// Mitsubishi GX Developer project: パレット移載装置   PLC: Q02

PROGRAM MAIN
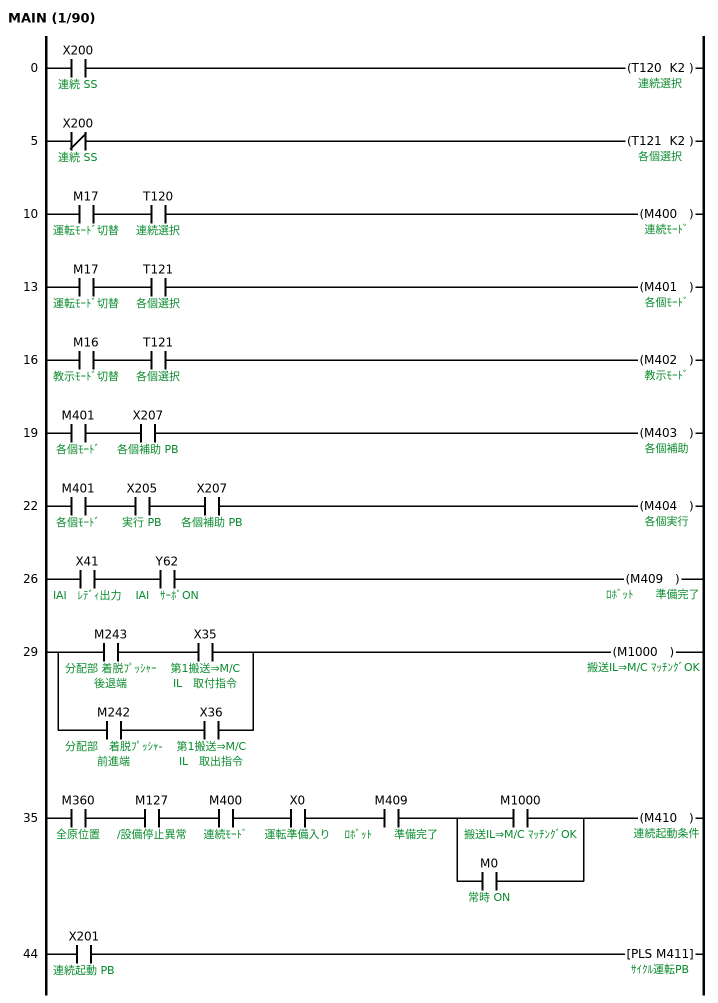
0     LD      X200  ; 連続 SS
      OUT     T120 K2  ; 連続選択
5     LDI     X200  ; 連続 SS
      OUT     T121 K2  ; 各個選択
10    LD      M17  ; 運転ﾓｰﾄﾞ切替
      AND     T120  ; 連続選択
      OUT     M400  ; 連続ﾓｰﾄﾞ
13    LD      M17  ; 運転ﾓｰﾄﾞ切替
      AND     T121  ; 各個選択
      OUT     M401  ; 各個ﾓｰﾄﾞ
16    LD      M16  ; 教示ﾓｰﾄﾞ切替
      AND     T121  ; 各個選択
      OUT     M402  ; 教示ﾓｰﾄﾞ
19    LD      M401  ; 各個ﾓｰﾄﾞ
      AND     X207  ; 各個補助 PB
      OUT     M403  ; 各個補助
22    LD      M401  ; 各個ﾓｰﾄﾞ
      AND     X205  ; 実行 PB
      AND     X207  ; 各個補助 PB
      OUT     M404  ; 各個実行
26    LD      X41  ; IAI　ﾚﾃﾞｨ出力
      AND     Y62  ; IAI　ｻｰﾎﾞON
      OUT     M409  ; ﾛﾎﾞｯﾄ　　準備完了
29    LD      M243  ; 分配部 着脱ﾌﾟｯｼｬｰ 後退端
      AND     X35  ; 第1搬送⇒M/C IL　取付指令
      LD      M242  ; 分配部　着脱ﾌﾟｯｼｬ- 前進端
      AND     X36  ; 第1搬送⇒M/C IL　取出指令
      ORB
      OUT     M1000  ; 搬送IL⇒M/C ﾏｯﾁﾝｸﾞOK
35    LD      M360  ; 全原位置
      AND     M127  ; /設備停止異常
      AND     M400  ; 連続ﾓｰﾄﾞ
      AND     X0  ; 運転準備入り
      AND     M409  ; ﾛﾎﾞｯﾄ　　準備完了
      LD      M1000  ; 搬送IL⇒M/C ﾏｯﾁﾝｸﾞOK
      OR      M0  ; 常時 ON
      ANB
      OUT     M410  ; 連続起動条件
44    LD      X201  ; 連続起動 PB
      PLS     M411  ; ｻｲｸﾙ運転PB
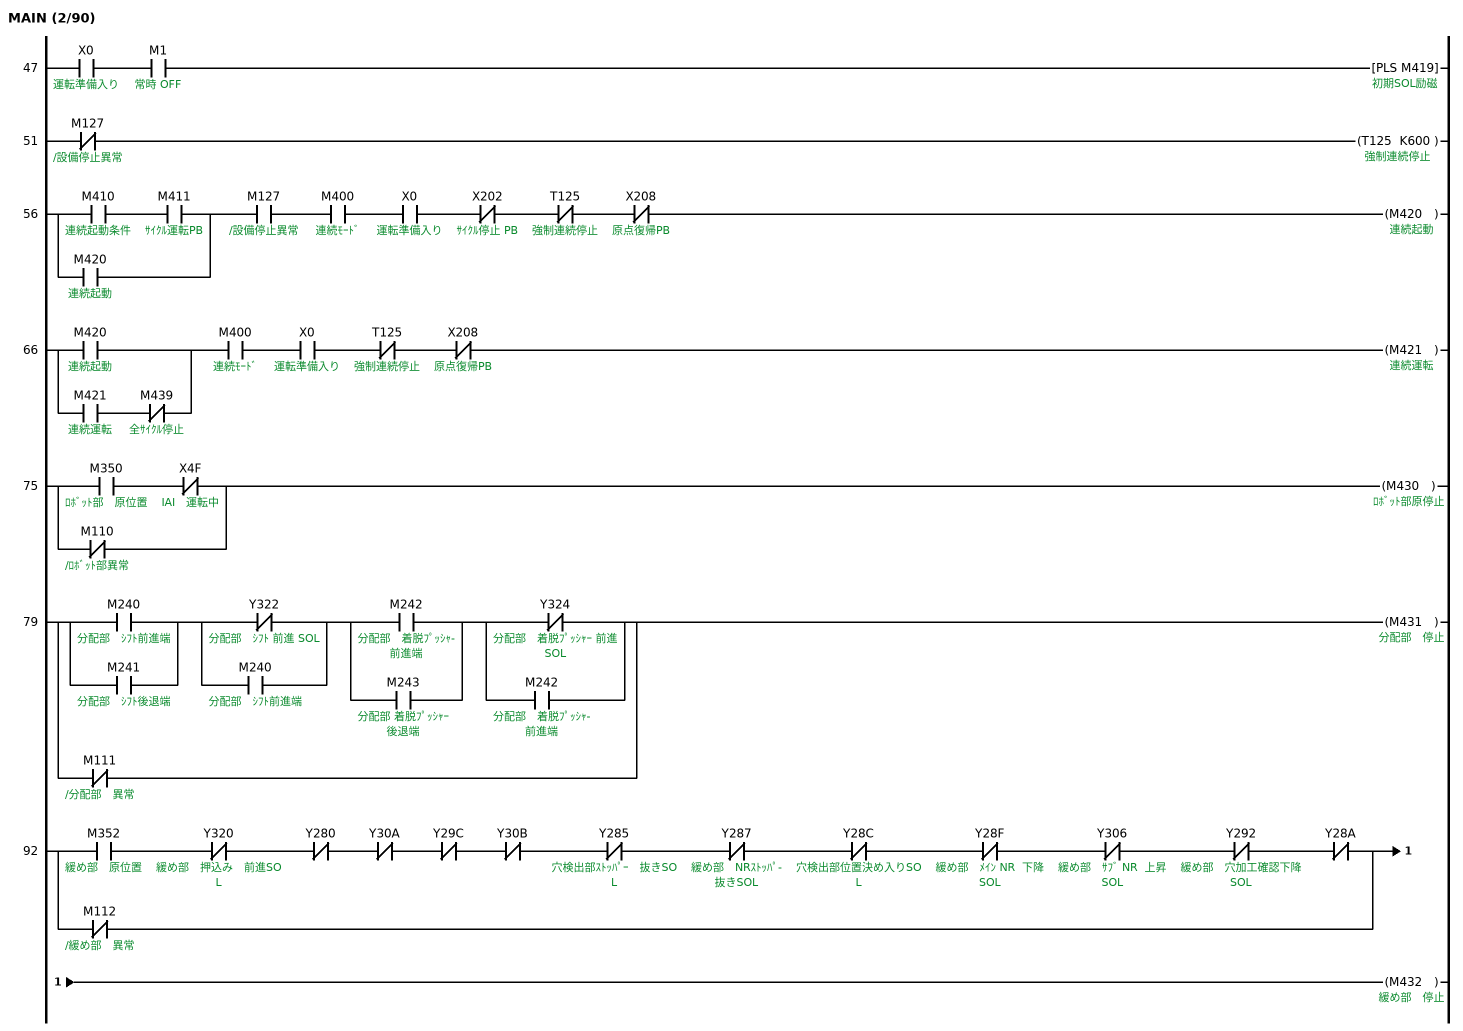
47    LD      X0  ; 運転準備入り
      AND     M1  ; 常時 OFF
      PLS     M419  ; 初期SOL励磁
51    LDI     M127  ; /設備停止異常
      OUT     T125 K600  ; 強制連続停止
56    LD      M410  ; 連続起動条件
      AND     M411  ; ｻｲｸﾙ運転PB
      OR      M420  ; 連続起動
      AND     M127  ; /設備停止異常
      AND     M400  ; 連続ﾓｰﾄﾞ
      AND     X0  ; 運転準備入り
      ANI     X202  ; ｻｲｸﾙ停止 PB
      ANI     T125  ; 強制連続停止
      ANI     X208  ; 原点復帰PB
      OUT     M420  ; 連続起動
66    LD      M420  ; 連続起動
      LD      M421  ; 連続運転
      ANI     M439  ; 全ｻｲｸﾙ停止
      ORB
      AND     M400  ; 連続ﾓｰﾄﾞ
      AND     X0  ; 運転準備入り
      ANI     T125  ; 強制連続停止
      ANI     X208  ; 原点復帰PB
      OUT     M421  ; 連続運転
75    LD      M350  ; ﾛﾎﾞｯﾄ部　原位置
      ANI     X4F  ; IAI　運転中
      ORI     M110  ; /ﾛﾎﾞｯﾄ部異常
      OUT     M430  ; ﾛﾎﾞｯﾄ部原停止
79    LD      M240  ; 分配部　ｼﾌﾄ前進端
      OR      M241  ; 分配部　ｼﾌﾄ後退端
      LDI     Y322  ; 分配部　ｼﾌﾄ 前進 SOL
      OR      M240  ; 分配部　ｼﾌﾄ前進端
      ANB
      LD      M242  ; 分配部　着脱ﾌﾟｯｼｬ- 前進端
      OR      M243  ; 分配部 着脱ﾌﾟｯｼｬｰ 後退端
      ANB
      LDI     Y324  ; 分配部　着脱ﾌﾟｯｼｬｰ 前進 SOL
      OR      M242  ; 分配部　着脱ﾌﾟｯｼｬ- 前進端
      ANB
      ORI     M111  ; /分配部　異常
      OUT     M431  ; 分配部　停止
92    LD      M352  ; 緩め部　原位置
      ANI     Y320  ; 緩め部　押込み　前進SOL
      ANI     Y280
      ANI     Y30A
      ANI     Y29C
      ANI     Y30B
      ANI     Y285  ; 穴検出部ｽﾄｯﾊﾟｰ　抜きSOL
      ANI     Y287  ; 緩め部　NRｽﾄｯﾊﾟ-抜きSOL
      ANI     Y28C  ; 穴検出部位置決め入りSOL
      ANI     Y28F  ; 緩め部　ﾒｲﾝ NR  下降 SOL
      ANI     Y306  ; 緩め部　ｻﾌﾞ NR  上昇 SOL
      ANI     Y292  ; 緩め部　穴加工確認下降 SOL
      ANI     Y28A
      ORI     M112  ; /緩め部　異常
      OUT     M432  ; 緩め部　停止
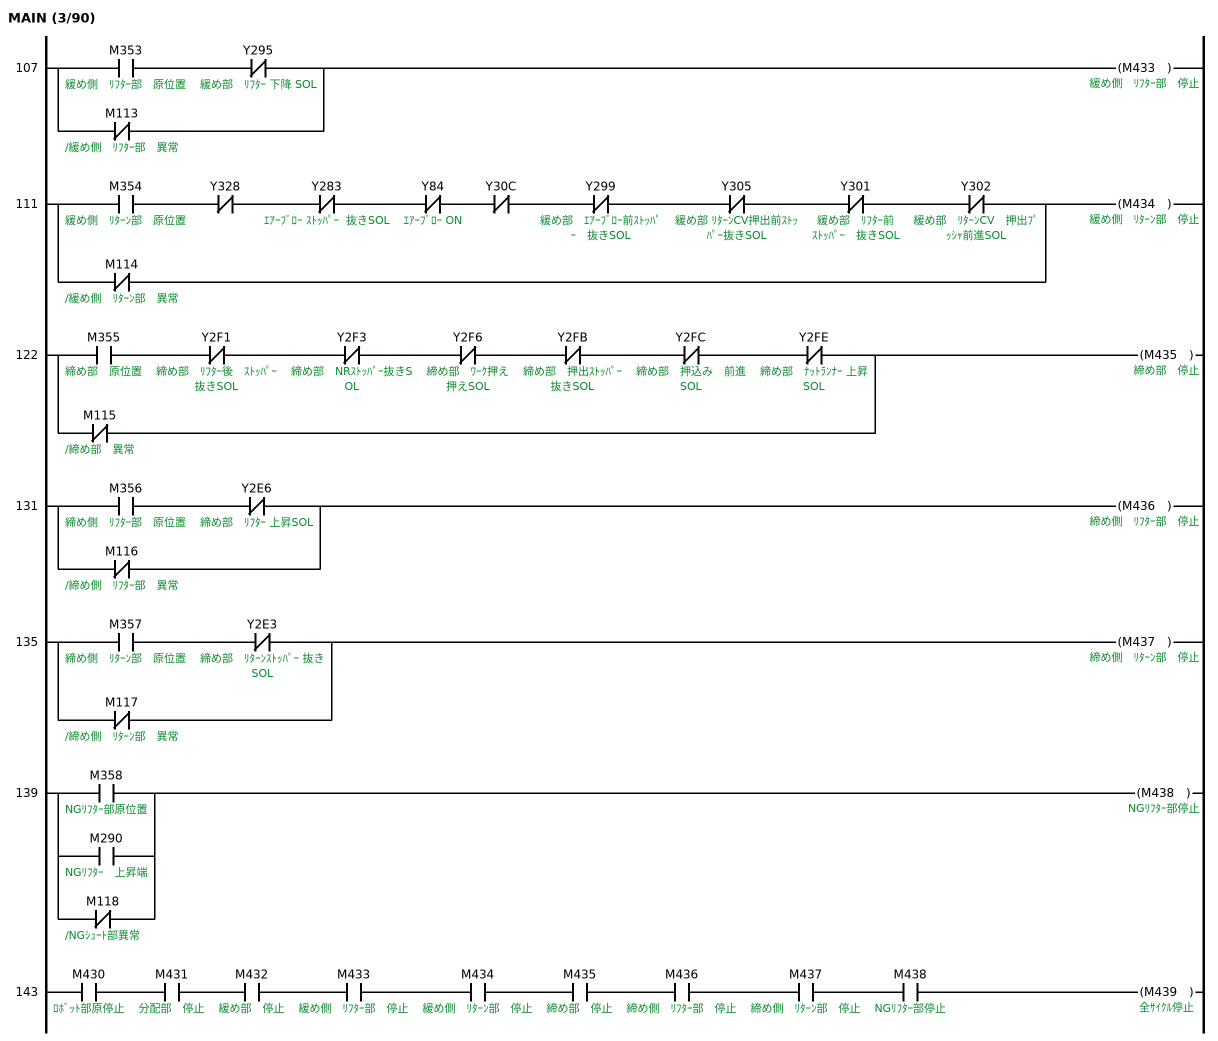
107   LD      M353  ; 緩め側　ﾘﾌﾀｰ部　原位置
      ANI     Y295  ; 緩め部　ﾘﾌﾀｰ 下降 SOL
      ORI     M113  ; /緩め側　ﾘﾌﾀｰ部　異常
      OUT     M433  ; 緩め側　ﾘﾌﾀｰ部　停止
111   LD      M354  ; 緩め側　ﾘﾀｰﾝ部　原位置
      ANI     Y328
      ANI     Y283  ; ｴｱｰﾌﾞﾛｰ ｽﾄｯﾊﾟｰ  抜きSOL
      ANI     Y84  ; ｴｱｰﾌﾞﾛｰ ON
      ANI     Y30C
      ANI     Y299  ; 緩め部　ｴｱｰﾌﾞﾛｰ前ｽﾄｯﾊﾟｰ　抜きSOL
      ANI     Y305  ; 緩め部 ﾘﾀｰﾝCV押出前ｽﾄｯﾊﾟｰ抜きSOL
      ANI     Y301  ; 緩め部　ﾘﾌﾀｰ前  ｽﾄｯﾊﾟｰ　抜きSOL
      ANI     Y302  ; 緩め部　ﾘﾀｰﾝCV　押出ﾌﾟｯｼｬ前進SOL
      ORI     M114  ; /緩め側　ﾘﾀｰﾝ部　異常
      OUT     M434  ; 緩め側　ﾘﾀｰﾝ部　停止
122   LD      M355  ; 締め部　原位置
      ANI     Y2F1  ; 締め部　ﾘﾌﾀｰ後　ｽﾄｯﾊﾟｰ　抜きSOL
      ANI     Y2F3  ; 締め部　NRｽﾄｯﾊﾟｰ抜きSOL
      ANI     Y2F6  ; 締め部　ﾜｰｸ押え 押えSOL
      ANI     Y2FB  ; 締め部　押出ｽﾄｯﾊﾟｰ 抜きSOL
      ANI     Y2FC  ; 締め部　押込み　前進 SOL
      ANI     Y2FE  ; 締め部　ﾅｯﾄﾗﾝﾅｰ 上昇 SOL
      ORI     M115  ; /締め部　異常
      OUT     M435  ; 締め部　停止
131   LD      M356  ; 締め側　ﾘﾌﾀｰ部　原位置
      ANI     Y2E6  ; 締め部　ﾘﾌﾀｰ 上昇SOL
      ORI     M116  ; /締め側　ﾘﾌﾀｰ部　異常
      OUT     M436  ; 締め側　ﾘﾌﾀｰ部　停止
135   LD      M357  ; 締め側　ﾘﾀｰﾝ部　原位置
      ANI     Y2E3  ; 締め部　ﾘﾀｰﾝｽﾄｯﾊﾟｰ 抜き SOL
      ORI     M117  ; /締め側　ﾘﾀｰﾝ部　異常
      OUT     M437  ; 締め側　ﾘﾀｰﾝ部　停止
139   LD      M358  ; NGﾘﾌﾀｰ部原位置
      OR      M290  ; NGﾘﾌﾀｰ　上昇端
      ORI     M118  ; /NGｼｭｰﾄ部異常
      OUT     M438  ; NGﾘﾌﾀｰ部停止
143   LD      M430  ; ﾛﾎﾞｯﾄ部原停止
      AND     M431  ; 分配部　停止
      AND     M432  ; 緩め部　停止
      AND     M433  ; 緩め側　ﾘﾌﾀｰ部　停止
      AND     M434  ; 緩め側　ﾘﾀｰﾝ部　停止
      AND     M435  ; 締め部　停止
      AND     M436  ; 締め側　ﾘﾌﾀｰ部　停止
      AND     M437  ; 締め側　ﾘﾀｰﾝ部　停止
      AND     M438  ; NGﾘﾌﾀｰ部停止
      OUT     M439  ; 全ｻｲｸﾙ停止
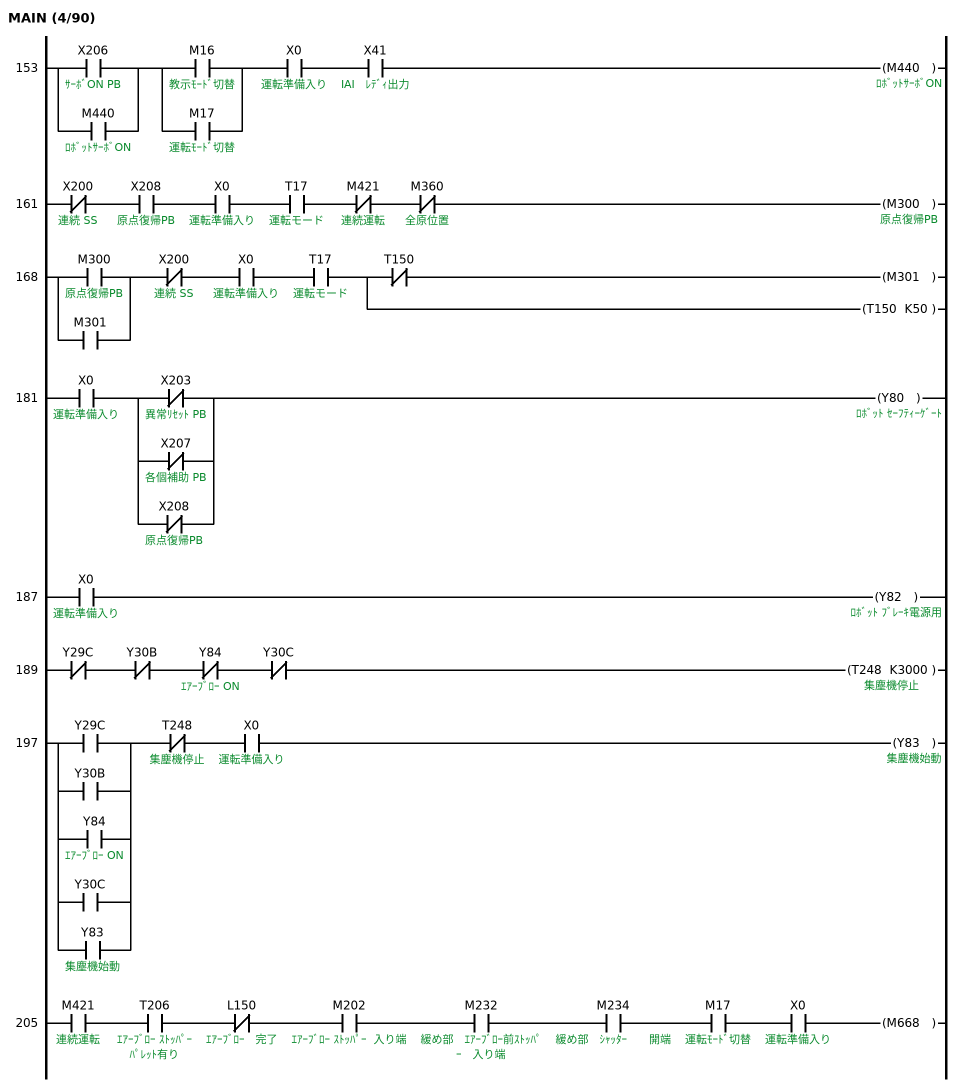
153   LD      X206  ; ｻｰﾎﾞON PB
      OR      M440  ; ﾛﾎﾞｯﾄｻｰﾎﾞON
      LD      M16  ; 教示ﾓｰﾄﾞ切替
      OR      M17  ; 運転ﾓｰﾄﾞ切替
      ANB
      AND     X0  ; 運転準備入り
      AND     X41  ; IAI　ﾚﾃﾞｨ出力
      OUT     M440  ; ﾛﾎﾞｯﾄｻｰﾎﾞON
161   LDI     X200  ; 連続 SS
      AND     X208  ; 原点復帰PB
      AND     X0  ; 運転準備入り
      AND     T17  ; 運転モード
      ANI     M421  ; 連続運転
      ANI     M360  ; 全原位置
      OUT     M300  ; 原点復帰PB
168   LD      M300  ; 原点復帰PB
      OR      M301
      ANI     X200  ; 連続 SS
      AND     X0  ; 運転準備入り
      AND     T17  ; 運転モード
      MPS
      ANI     T150
      OUT     M301
      MPP
      OUT     T150 K50
181   LD      X0  ; 運転準備入り
      LDI     X203  ; 異常ﾘｾｯﾄ PB
      ORI     X207  ; 各個補助 PB
      ORI     X208  ; 原点復帰PB
      ANB
      OUT     Y80  ; ﾛﾎﾞｯﾄ ｾｰﾌﾃｨｰｹﾞｰﾄ
187   LD      X0  ; 運転準備入り
      OUT     Y82  ; ﾛﾎﾞｯﾄ ﾌﾞﾚｰｷ電源用
189   LDI     Y29C
      ANI     Y30B
      ANI     Y84  ; ｴｱｰﾌﾞﾛｰ ON
      ANI     Y30C
      OUT     T248 K3000  ; 集塵機停止
197   LD      Y29C
      OR      Y30B
      OR      Y84  ; ｴｱｰﾌﾞﾛｰ ON
      OR      Y30C
      OR      Y83  ; 集塵機始動
      ANI     T248  ; 集塵機停止
      AND     X0  ; 運転準備入り
      OUT     Y83  ; 集塵機始動
205   LD      M421  ; 連続運転
      AND     T206  ; ｴｱｰﾌﾞﾛｰ ｽﾄｯﾊﾟｰ  ﾊﾟﾚｯﾄ有り
      ANI     L150  ; ｴｱｰﾌﾞﾛｰ　完了
      AND     M202  ; ｴｱｰﾌﾞﾛｰ ｽﾄｯﾊﾟｰ  入り端
      AND     M232  ; 緩め部　ｴｱｰﾌﾞﾛｰ前ｽﾄｯﾊﾟｰ　入り端
      AND     M234  ; 緩め部　ｼｬｯﾀｰ　　開端
      AND     M17  ; 運転ﾓｰﾄﾞ切替
      AND     X0  ; 運転準備入り
      OUT     M668
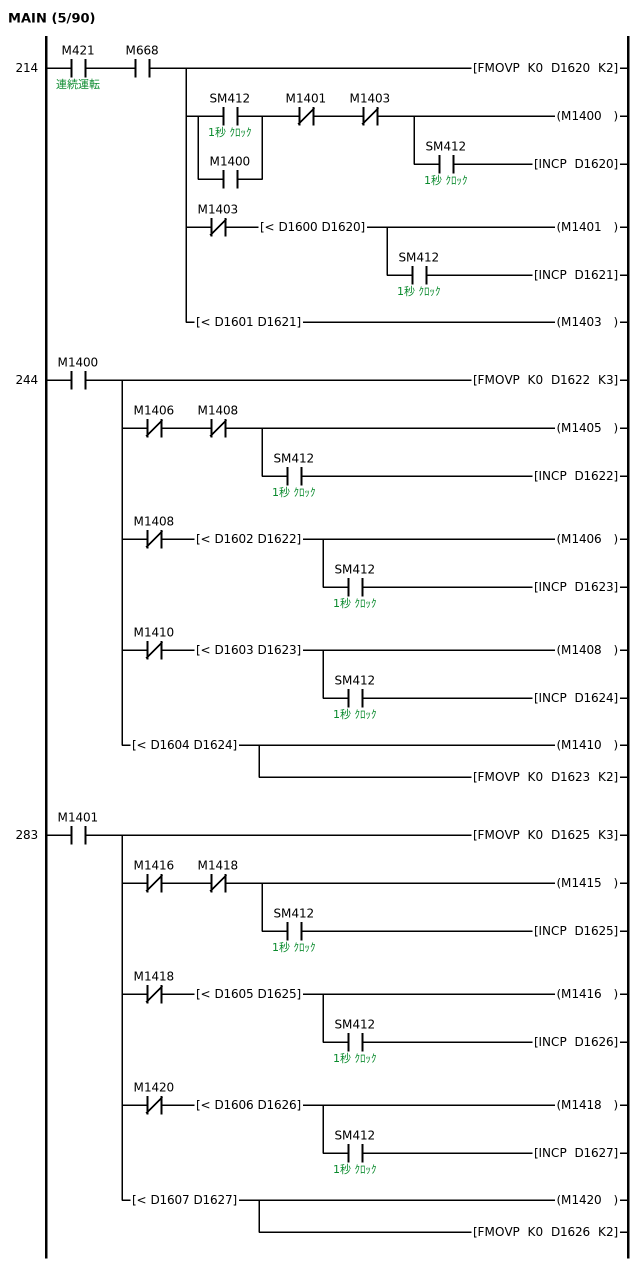
214   LD      M421  ; 連続運転
      AND     M668
      FMOVP   K0 D1620 K2
      MPS
      LD      SM412  ; 1秒 ｸﾛｯｸ
      OR      M1400
      ANB
      ANI     M1401
      ANI     M1403
      OUT     M1400
      AND     SM412  ; 1秒 ｸﾛｯｸ
      INCP    D1620
      MRD
      ANI     M1403
      AND<    D1600 D1620
      OUT     M1401
      AND     SM412  ; 1秒 ｸﾛｯｸ
      INCP    D1621
      MPP
      AND<    D1601 D1621
      OUT     M1403
244   LD      M1400
      FMOVP   K0 D1622 K3
      MPS
      ANI     M1406
      ANI     M1408
      OUT     M1405
      AND     SM412  ; 1秒 ｸﾛｯｸ
      INCP    D1622
      MRD
      ANI     M1408
      AND<    D1602 D1622
      OUT     M1406
      AND     SM412  ; 1秒 ｸﾛｯｸ
      INCP    D1623
      MRD
      ANI     M1410
      AND<    D1603 D1623
      OUT     M1408
      AND     SM412  ; 1秒 ｸﾛｯｸ
      INCP    D1624
      MPP
      AND<    D1604 D1624
      OUT     M1410
      FMOVP   K0 D1623 K2
283   LD      M1401
      FMOVP   K0 D1625 K3
      MPS
      ANI     M1416
      ANI     M1418
      OUT     M1415
      AND     SM412  ; 1秒 ｸﾛｯｸ
      INCP    D1625
      MRD
      ANI     M1418
      AND<    D1605 D1625
      OUT     M1416
      AND     SM412  ; 1秒 ｸﾛｯｸ
      INCP    D1626
      MRD
      ANI     M1420
      AND<    D1606 D1626
      OUT     M1418
      AND     SM412  ; 1秒 ｸﾛｯｸ
      INCP    D1627
      MPP
      AND<    D1607 D1627
      OUT     M1420
      FMOVP   K0 D1626 K2
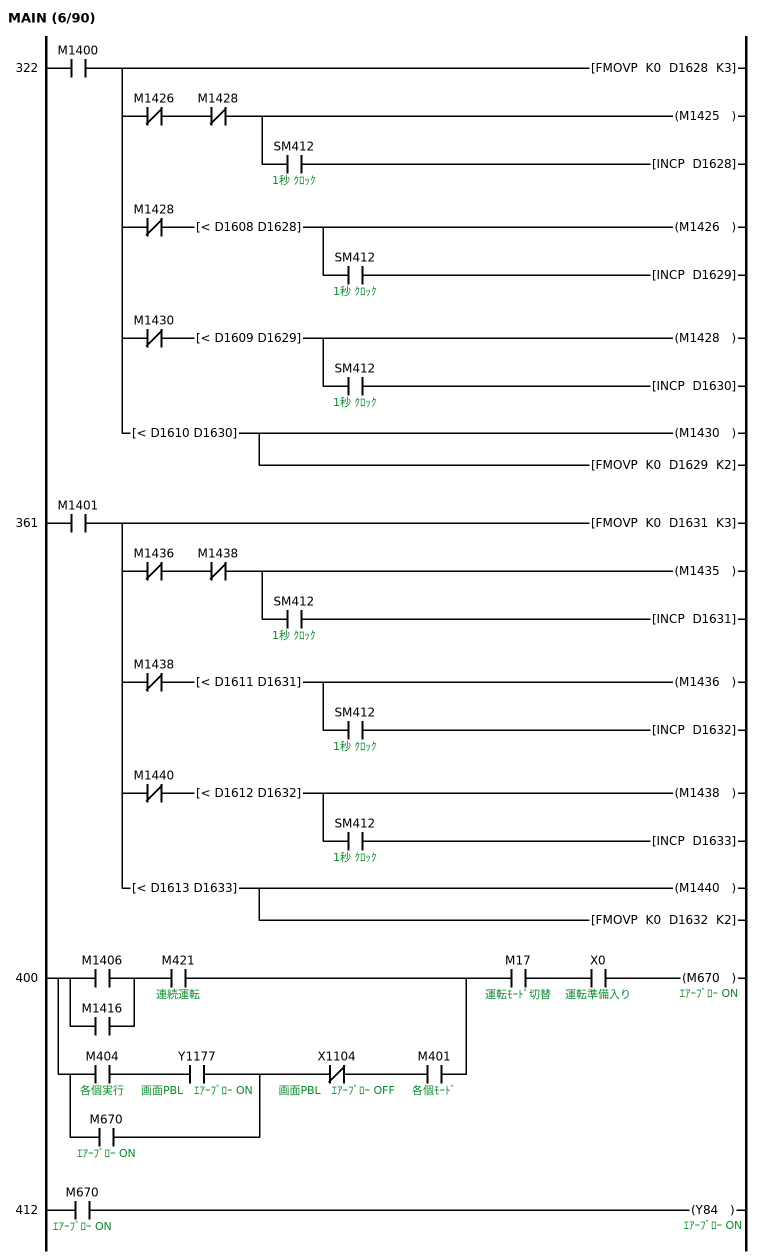
322   LD      M1400
      FMOVP   K0 D1628 K3
      MPS
      ANI     M1426
      ANI     M1428
      OUT     M1425
      AND     SM412  ; 1秒 ｸﾛｯｸ
      INCP    D1628
      MRD
      ANI     M1428
      AND<    D1608 D1628
      OUT     M1426
      AND     SM412  ; 1秒 ｸﾛｯｸ
      INCP    D1629
      MRD
      ANI     M1430
      AND<    D1609 D1629
      OUT     M1428
      AND     SM412  ; 1秒 ｸﾛｯｸ
      INCP    D1630
      MPP
      AND<    D1610 D1630
      OUT     M1430
      FMOVP   K0 D1629 K2
361   LD      M1401
      FMOVP   K0 D1631 K3
      MPS
      ANI     M1436
      ANI     M1438
      OUT     M1435
      AND     SM412  ; 1秒 ｸﾛｯｸ
      INCP    D1631
      MRD
      ANI     M1438
      AND<    D1611 D1631
      OUT     M1436
      AND     SM412  ; 1秒 ｸﾛｯｸ
      INCP    D1632
      MRD
      ANI     M1440
      AND<    D1612 D1632
      OUT     M1438
      AND     SM412  ; 1秒 ｸﾛｯｸ
      INCP    D1633
      MPP
      AND<    D1613 D1633
      OUT     M1440
      FMOVP   K0 D1632 K2
400   LD      M1406
      OR      M1416
      AND     M421  ; 連続運転
      LD      M404  ; 各個実行
      AND     Y1177  ; 画面PBL　ｴｱｰﾌﾞﾛｰ ON
      OR      M670  ; ｴｱｰﾌﾞﾛｰ ON
      ANI     X1104  ; 画面PBL　ｴｱｰﾌﾞﾛｰ OFF
      AND     M401  ; 各個ﾓｰﾄﾞ
      ORB
      AND     M17  ; 運転ﾓｰﾄﾞ切替
      AND     X0  ; 運転準備入り
      OUT     M670  ; ｴｱｰﾌﾞﾛｰ ON
412   LD      M670  ; ｴｱｰﾌﾞﾛｰ ON
      OUT     Y84  ; ｴｱｰﾌﾞﾛｰ ON
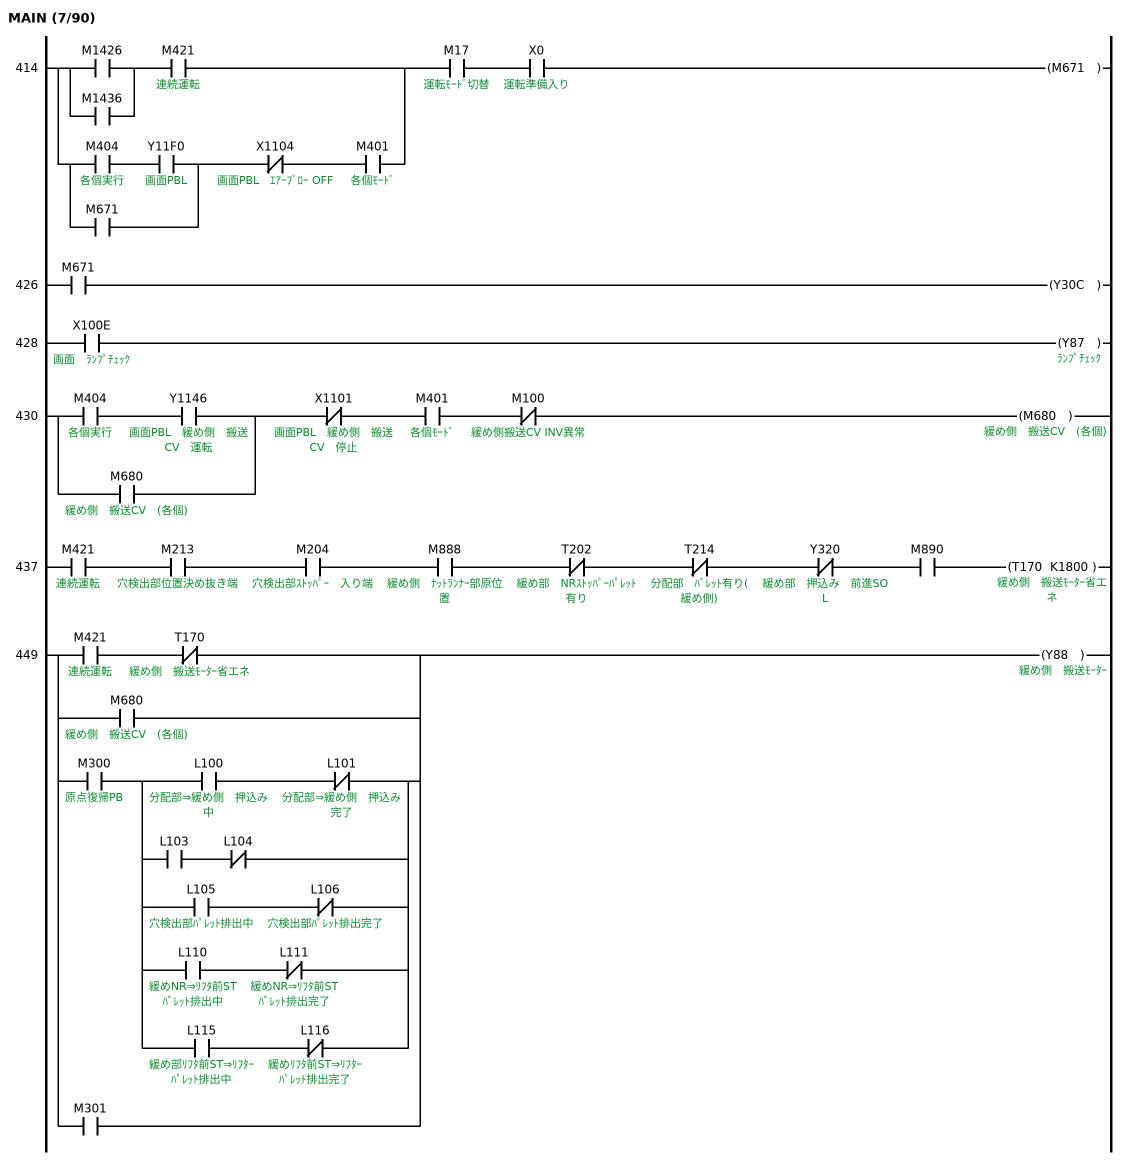
414   LD      M1426
      OR      M1436
      AND     M421  ; 連続運転
      LD      M404  ; 各個実行
      AND     Y11F0  ; 画面PBL
      OR      M671
      ANI     X1104  ; 画面PBL　ｴｱｰﾌﾞﾛｰ OFF
      AND     M401  ; 各個ﾓｰﾄﾞ
      ORB
      AND     M17  ; 運転ﾓｰﾄﾞ切替
      AND     X0  ; 運転準備入り
      OUT     M671
426   LD      M671
      OUT     Y30C
428   LD      X100E  ; 画面　ﾗﾝﾌﾟﾁｪｯｸ
      OUT     Y87  ; ﾗﾝﾌﾟﾁｪｯｸ
430   LD      M404  ; 各個実行
      AND     Y1146  ; 画面PBL　緩め側　搬送CV　運転
      OR      M680  ; 緩め側　搬送CV　(各個)
      ANI     X1101  ; 画面PBL　緩め側　搬送CV　停止
      AND     M401  ; 各個ﾓｰﾄﾞ
      ANI     M100  ; 緩め側搬送CV INV異常
      OUT     M680  ; 緩め側　搬送CV　(各個)
437   LD      M421  ; 連続運転
      AND     M213  ; 穴検出部位置決め抜き端
      AND     M204  ; 穴検出部ｽﾄｯﾊﾟｰ　入り端
      AND     M888  ; 緩め側　ﾅｯﾄﾗﾝﾅｰ部原位置
      ANI     T202  ; 緩め部　NRｽﾄｯﾊﾟｰﾊﾟﾚｯﾄ有り
      ANI     T214  ; 分配部　ﾊﾟﾚｯﾄ有り(緩め側)
      ANI     Y320  ; 緩め部　押込み　前進SOL
      AND     M890
      OUT     T170 K1800  ; 緩め側　搬送ﾓｰﾀｰ省エネ
449   LD      M421  ; 連続運転
      ANI     T170  ; 緩め側　搬送ﾓｰﾀｰ省エネ
      OR      M680  ; 緩め側　搬送CV　(各個)
      LD      M300  ; 原点復帰PB
      LD      L100  ; 分配部⇒緩め側　押込み中
      ANI     L101  ; 分配部⇒緩め側　押込み完了
      LD      L103
      ANI     L104
      ORB
      LD      L105  ; 穴検出部ﾊﾟﾚｯﾄ排出中
      ANI     L106  ; 穴検出部ﾊﾟﾚｯﾄ排出完了
      ORB
      LD      L110  ; 緩めNR⇒ﾘﾌﾀ前ST ﾊﾟﾚｯﾄ排出中
      ANI     L111  ; 緩めNR⇒ﾘﾌﾀ前ST ﾊﾟﾚｯﾄ排出完了
      ORB
      LD      L115  ; 緩め部ﾘﾌﾀ前ST⇒ﾘﾌﾀｰ ﾊﾟﾚｯﾄ排出中
      ANI     L116  ; 緩めﾘﾌﾀ前ST⇒ﾘﾌﾀｰ ﾊﾟﾚｯﾄ排出完了
      ORB
      ANB
      ORB
      OR      M301
      OUT     Y88  ; 緩め側　搬送ﾓｰﾀｰ
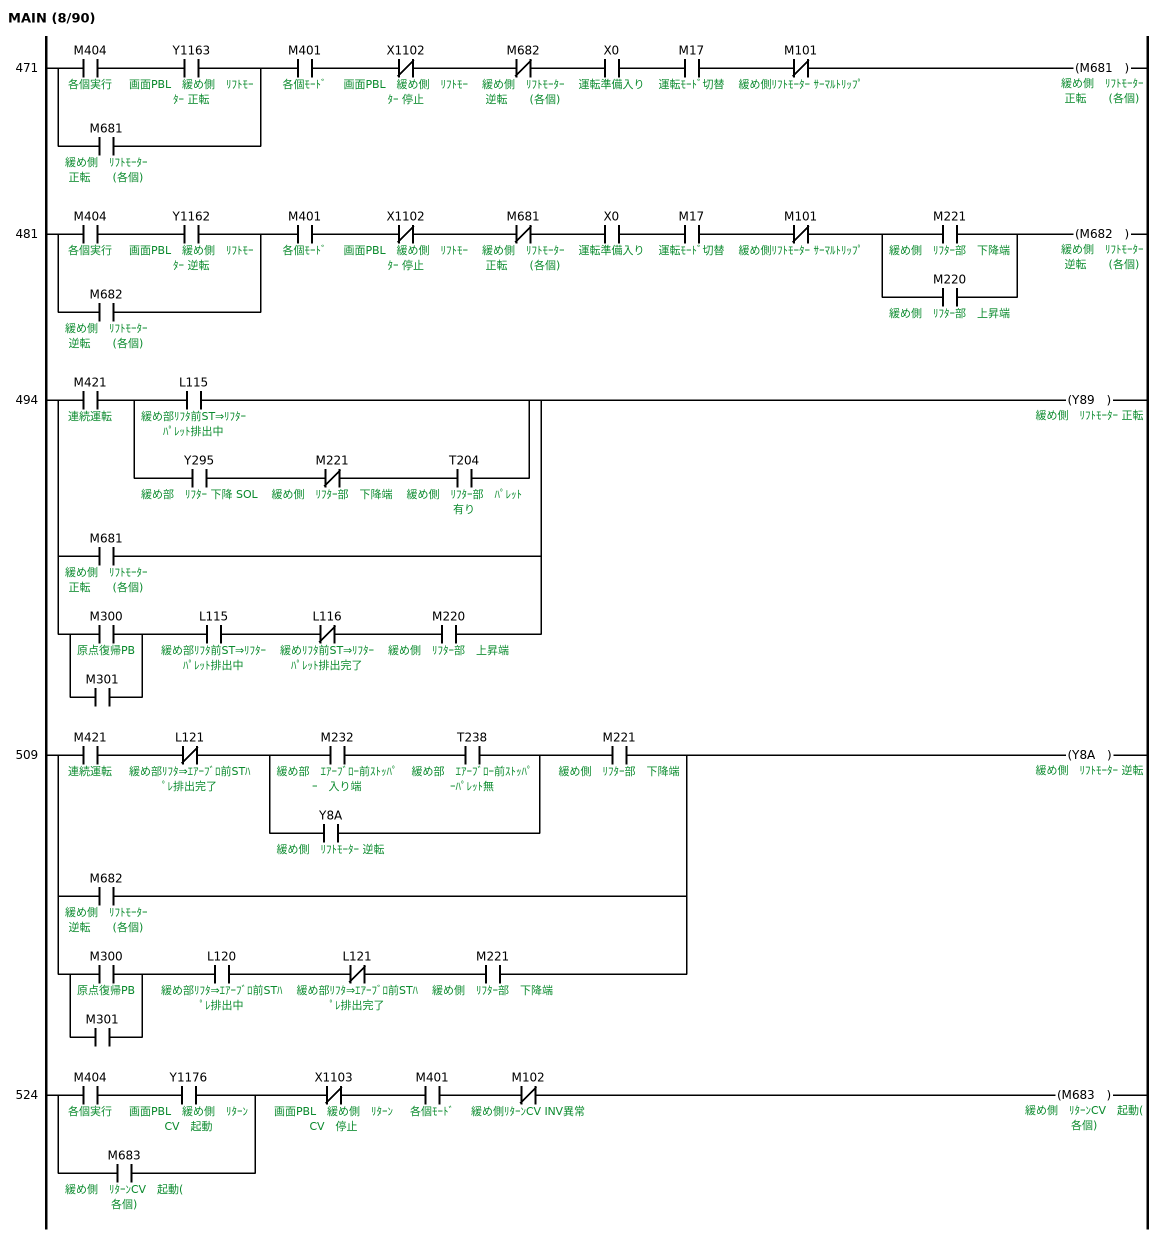
471   LD      M404  ; 各個実行
      AND     Y1163  ; 画面PBL　緩め側　ﾘﾌﾄﾓｰﾀｰ 正転
      OR      M681  ; 緩め側　ﾘﾌﾄﾓｰﾀｰ 正転　　(各個)
      AND     M401  ; 各個ﾓｰﾄﾞ
      ANI     X1102  ; 画面PBL　緩め側　ﾘﾌﾄﾓｰﾀｰ 停止
      ANI     M682  ; 緩め側　ﾘﾌﾄﾓｰﾀｰ 逆転　　(各個)
      AND     X0  ; 運転準備入り
      AND     M17  ; 運転ﾓｰﾄﾞ切替
      ANI     M101  ; 緩め側ﾘﾌﾄﾓｰﾀｰ ｻｰﾏﾙﾄﾘｯﾌﾟ
      OUT     M681  ; 緩め側　ﾘﾌﾄﾓｰﾀｰ 正転　　(各個)
481   LD      M404  ; 各個実行
      AND     Y1162  ; 画面PBL　緩め側　ﾘﾌﾄﾓｰﾀｰ 逆転
      OR      M682  ; 緩め側　ﾘﾌﾄﾓｰﾀｰ 逆転　　(各個)
      AND     M401  ; 各個ﾓｰﾄﾞ
      ANI     X1102  ; 画面PBL　緩め側　ﾘﾌﾄﾓｰﾀｰ 停止
      ANI     M681  ; 緩め側　ﾘﾌﾄﾓｰﾀｰ 正転　　(各個)
      AND     X0  ; 運転準備入り
      AND     M17  ; 運転ﾓｰﾄﾞ切替
      ANI     M101  ; 緩め側ﾘﾌﾄﾓｰﾀｰ ｻｰﾏﾙﾄﾘｯﾌﾟ
      LD      M221  ; 緩め側　ﾘﾌﾀｰ部　下降端
      OR      M220  ; 緩め側　ﾘﾌﾀｰ部　上昇端
      ANB
      OUT     M682  ; 緩め側　ﾘﾌﾄﾓｰﾀｰ 逆転　　(各個)
494   LD      M421  ; 連続運転
      LD      L115  ; 緩め部ﾘﾌﾀ前ST⇒ﾘﾌﾀｰ ﾊﾟﾚｯﾄ排出中
      LD      Y295  ; 緩め部　ﾘﾌﾀｰ 下降 SOL
      ANI     M221  ; 緩め側　ﾘﾌﾀｰ部　下降端
      AND     T204  ; 緩め側　ﾘﾌﾀｰ部　ﾊﾟﾚｯﾄ有り
      ORB
      ANB
      OR      M681  ; 緩め側　ﾘﾌﾄﾓｰﾀｰ 正転　　(各個)
      LD      M300  ; 原点復帰PB
      OR      M301
      AND     L115  ; 緩め部ﾘﾌﾀ前ST⇒ﾘﾌﾀｰ ﾊﾟﾚｯﾄ排出中
      ANI     L116  ; 緩めﾘﾌﾀ前ST⇒ﾘﾌﾀｰ ﾊﾟﾚｯﾄ排出完了
      AND     M220  ; 緩め側　ﾘﾌﾀｰ部　上昇端
      ORB
      OUT     Y89  ; 緩め側　ﾘﾌﾄﾓｰﾀｰ 正転
509   LD      M421  ; 連続運転
      ANI     L121  ; 緩め部ﾘﾌﾀ⇒ｴｱｰﾌﾞﾛ前STﾊﾟﾚ排出完了
      LD      M232  ; 緩め部　ｴｱｰﾌﾞﾛｰ前ｽﾄｯﾊﾟｰ　入り端
      AND     T238  ; 緩め部　ｴｱｰﾌﾞﾛｰ前ｽﾄｯﾊﾟｰﾊﾟﾚｯﾄ無
      OR      Y8A  ; 緩め側　ﾘﾌﾄﾓｰﾀｰ 逆転
      ANB
      AND     M221  ; 緩め側　ﾘﾌﾀｰ部　下降端
      OR      M682  ; 緩め側　ﾘﾌﾄﾓｰﾀｰ 逆転　　(各個)
      LD      M300  ; 原点復帰PB
      OR      M301
      AND     L120  ; 緩め部ﾘﾌﾀ⇒ｴｱｰﾌﾞﾛ前STﾊﾟﾚ排出中
      ANI     L121  ; 緩め部ﾘﾌﾀ⇒ｴｱｰﾌﾞﾛ前STﾊﾟﾚ排出完了
      AND     M221  ; 緩め側　ﾘﾌﾀｰ部　下降端
      ORB
      OUT     Y8A  ; 緩め側　ﾘﾌﾄﾓｰﾀｰ 逆転
524   LD      M404  ; 各個実行
      AND     Y1176  ; 画面PBL　緩め側　ﾘﾀｰﾝCV　起動
      OR      M683  ; 緩め側　ﾘﾀｰﾝCV　起動(各個)
      ANI     X1103  ; 画面PBL　緩め側　ﾘﾀｰﾝCV　停止
      AND     M401  ; 各個ﾓｰﾄﾞ
      ANI     M102  ; 緩め側ﾘﾀｰﾝCV INV異常
      OUT     M683  ; 緩め側　ﾘﾀｰﾝCV　起動(各個)
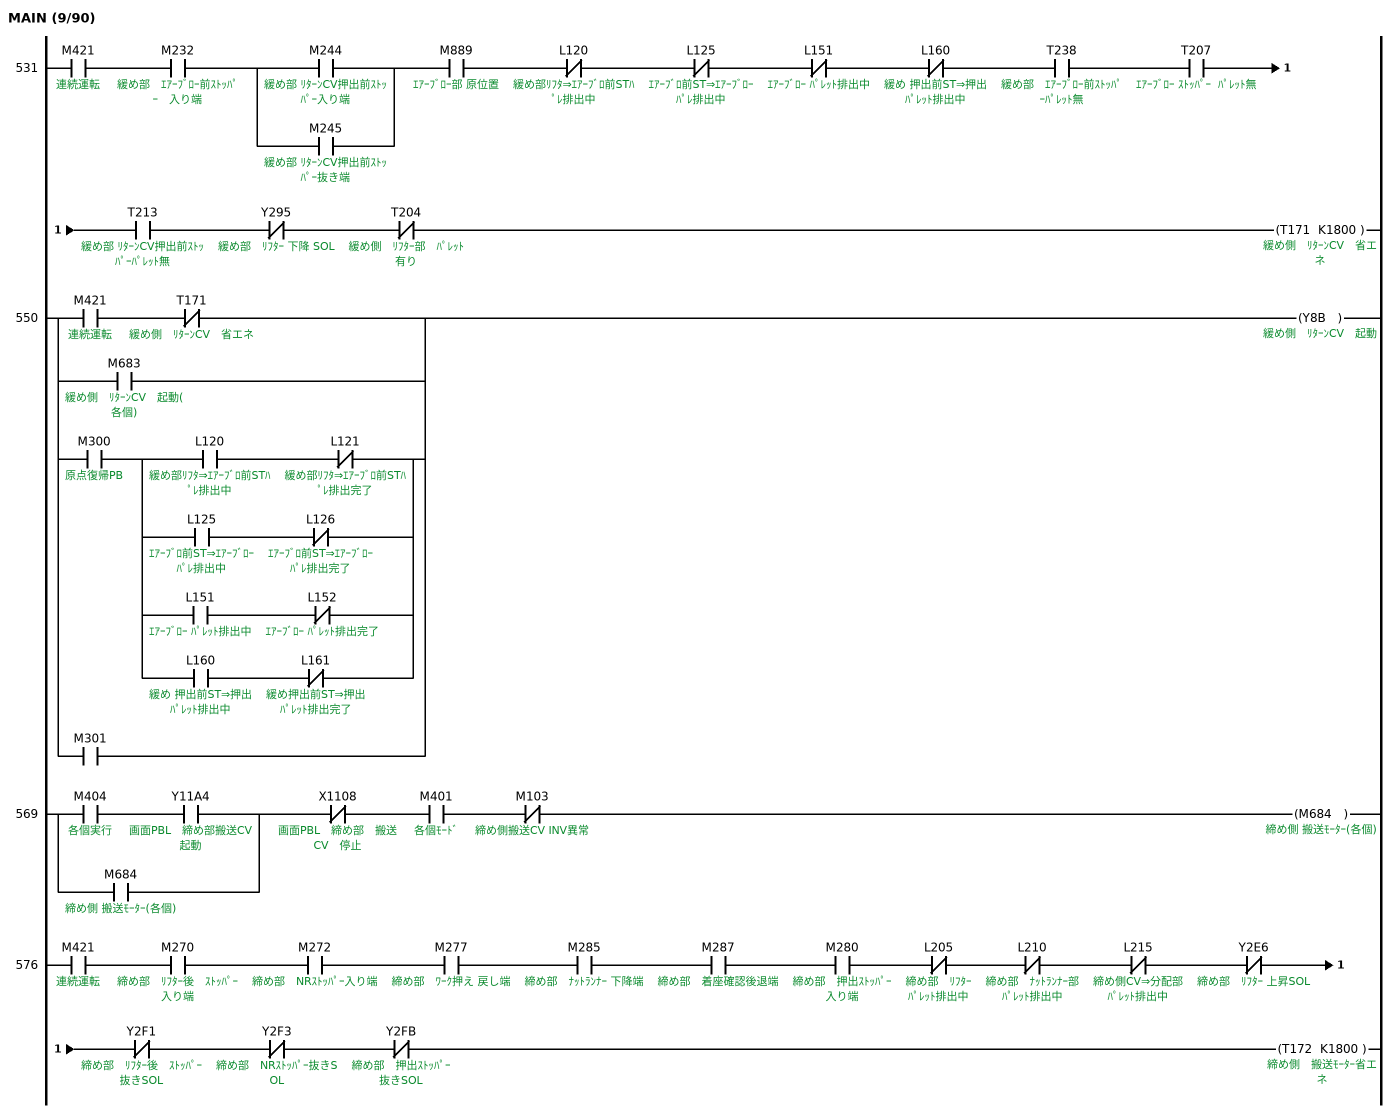
531   LD      M421  ; 連続運転
      AND     M232  ; 緩め部　ｴｱｰﾌﾞﾛｰ前ｽﾄｯﾊﾟｰ　入り端
      LD      M244  ; 緩め部 ﾘﾀｰﾝCV押出前ｽﾄｯﾊﾟｰ入り端
      OR      M245  ; 緩め部 ﾘﾀｰﾝCV押出前ｽﾄｯﾊﾟｰ抜き端
      ANB
      AND     M889  ; ｴｱｰﾌﾞﾛｰ部 原位置
      ANI     L120  ; 緩め部ﾘﾌﾀ⇒ｴｱｰﾌﾞﾛ前STﾊﾟﾚ排出中
      ANI     L125  ; ｴｱｰﾌﾞﾛ前ST⇒ｴｱｰﾌﾞﾛｰ ﾊﾟﾚ排出中
      ANI     L151  ; ｴｱｰﾌﾞﾛｰ ﾊﾟﾚｯﾄ排出中
      ANI     L160  ; 緩め 押出前ST⇒押出 ﾊﾟﾚｯﾄ排出中
      AND     T238  ; 緩め部　ｴｱｰﾌﾞﾛｰ前ｽﾄｯﾊﾟｰﾊﾟﾚｯﾄ無
      AND     T207  ; ｴｱｰﾌﾞﾛｰ ｽﾄｯﾊﾟｰ  ﾊﾟﾚｯﾄ無
      AND     T213  ; 緩め部 ﾘﾀｰﾝCV押出前ｽﾄｯﾊﾟｰﾊﾟﾚｯﾄ無
      ANI     Y295  ; 緩め部　ﾘﾌﾀｰ 下降 SOL
      ANI     T204  ; 緩め側　ﾘﾌﾀｰ部　ﾊﾟﾚｯﾄ有り
      OUT     T171 K1800  ; 緩め側　ﾘﾀｰﾝCV　省エネ
550   LD      M421  ; 連続運転
      ANI     T171  ; 緩め側　ﾘﾀｰﾝCV　省エネ
      OR      M683  ; 緩め側　ﾘﾀｰﾝCV　起動(各個)
      LD      M300  ; 原点復帰PB
      LD      L120  ; 緩め部ﾘﾌﾀ⇒ｴｱｰﾌﾞﾛ前STﾊﾟﾚ排出中
      ANI     L121  ; 緩め部ﾘﾌﾀ⇒ｴｱｰﾌﾞﾛ前STﾊﾟﾚ排出完了
      LD      L125  ; ｴｱｰﾌﾞﾛ前ST⇒ｴｱｰﾌﾞﾛｰ ﾊﾟﾚ排出中
      ANI     L126  ; ｴｱｰﾌﾞﾛ前ST⇒ｴｱｰﾌﾞﾛｰ ﾊﾟﾚ排出完了
      ORB
      LD      L151  ; ｴｱｰﾌﾞﾛｰ ﾊﾟﾚｯﾄ排出中
      ANI     L152  ; ｴｱｰﾌﾞﾛｰ ﾊﾟﾚｯﾄ排出完了
      ORB
      LD      L160  ; 緩め 押出前ST⇒押出 ﾊﾟﾚｯﾄ排出中
      ANI     L161  ; 緩め押出前ST⇒押出 ﾊﾟﾚｯﾄ排出完了
      ORB
      ANB
      ORB
      OR      M301
      OUT     Y8B  ; 緩め側　ﾘﾀｰﾝCV　起動
569   LD      M404  ; 各個実行
      AND     Y11A4  ; 画面PBL　締め部搬送CV起動
      OR      M684  ; 締め側 搬送ﾓｰﾀｰ(各個)
      ANI     X1108  ; 画面PBL　締め部　搬送CV　停止
      AND     M401  ; 各個ﾓｰﾄﾞ
      ANI     M103  ; 締め側搬送CV INV異常
      OUT     M684  ; 締め側 搬送ﾓｰﾀｰ(各個)
576   LD      M421  ; 連続運転
      AND     M270  ; 締め部　ﾘﾌﾀｰ後　ｽﾄｯﾊﾟｰ　入り端
      AND     M272  ; 締め部　NRｽﾄｯﾊﾟｰ入り端
      AND     M277  ; 締め部　ﾜｰｸ押え 戻し端
      AND     M285  ; 締め部　ﾅｯﾄﾗﾝﾅｰ 下降端
      AND     M287  ; 締め部　着座確認後退端
      AND     M280  ; 締め部　押出ｽﾄｯﾊﾟｰ 入り端
      ANI     L205  ; 締め部　ﾘﾌﾀｰ ﾊﾟﾚｯﾄ排出中
      ANI     L210  ; 締め部　ﾅｯﾄﾗﾝﾅｰ部 ﾊﾟﾚｯﾄ排出中
      ANI     L215  ; 締め側CV⇒分配部 ﾊﾟﾚｯﾄ排出中
      ANI     Y2E6  ; 締め部　ﾘﾌﾀｰ 上昇SOL
      ANI     Y2F1  ; 締め部　ﾘﾌﾀｰ後　ｽﾄｯﾊﾟｰ　抜きSOL
      ANI     Y2F3  ; 締め部　NRｽﾄｯﾊﾟｰ抜きSOL
      ANI     Y2FB  ; 締め部　押出ｽﾄｯﾊﾟｰ 抜きSOL
      OUT     T172 K1800  ; 締め側　搬送ﾓｰﾀｰ省エネ
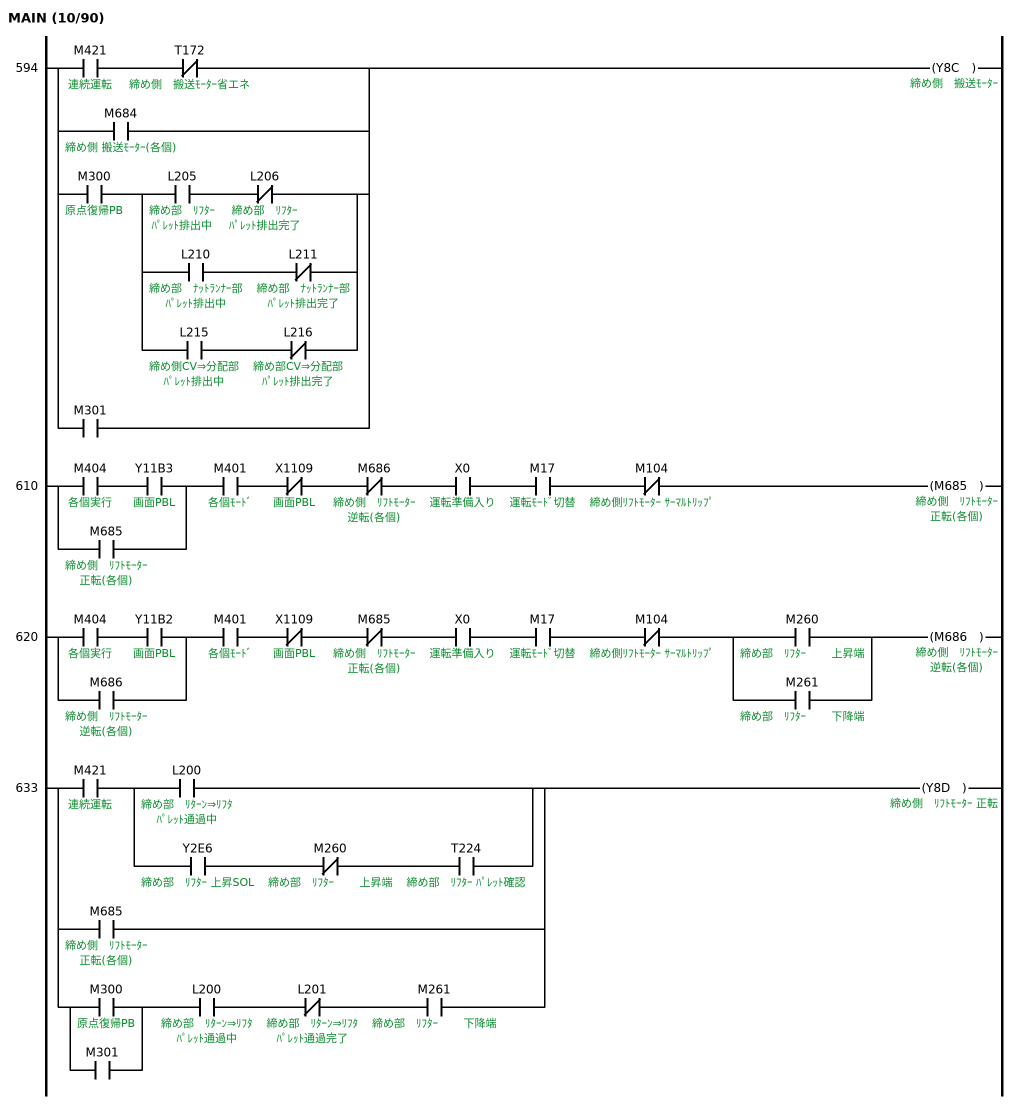
594   LD      M421  ; 連続運転
      ANI     T172  ; 締め側　搬送ﾓｰﾀｰ省エネ
      OR      M684  ; 締め側 搬送ﾓｰﾀｰ(各個)
      LD      M300  ; 原点復帰PB
      LD      L205  ; 締め部　ﾘﾌﾀｰ ﾊﾟﾚｯﾄ排出中
      ANI     L206  ; 締め部　ﾘﾌﾀｰ ﾊﾟﾚｯﾄ排出完了
      LD      L210  ; 締め部　ﾅｯﾄﾗﾝﾅｰ部 ﾊﾟﾚｯﾄ排出中
      ANI     L211  ; 締め部　ﾅｯﾄﾗﾝﾅｰ部 ﾊﾟﾚｯﾄ排出完了
      ORB
      LD      L215  ; 締め側CV⇒分配部 ﾊﾟﾚｯﾄ排出中
      ANI     L216  ; 締め部CV⇒分配部 ﾊﾟﾚｯﾄ排出完了
      ORB
      ANB
      ORB
      OR      M301
      OUT     Y8C  ; 締め側　搬送ﾓｰﾀｰ
610   LD      M404  ; 各個実行
      AND     Y11B3  ; 画面PBL
      OR      M685  ; 締め側　ﾘﾌﾄﾓｰﾀｰ 正転(各個)
      AND     M401  ; 各個ﾓｰﾄﾞ
      ANI     X1109  ; 画面PBL
      ANI     M686  ; 締め側　ﾘﾌﾄﾓｰﾀｰ 逆転(各個)
      AND     X0  ; 運転準備入り
      AND     M17  ; 運転ﾓｰﾄﾞ切替
      ANI     M104  ; 締め側ﾘﾌﾄﾓｰﾀｰ ｻｰﾏﾙﾄﾘｯﾌﾟ
      OUT     M685  ; 締め側　ﾘﾌﾄﾓｰﾀｰ 正転(各個)
620   LD      M404  ; 各個実行
      AND     Y11B2  ; 画面PBL
      OR      M686  ; 締め側　ﾘﾌﾄﾓｰﾀｰ 逆転(各個)
      AND     M401  ; 各個ﾓｰﾄﾞ
      ANI     X1109  ; 画面PBL
      ANI     M685  ; 締め側　ﾘﾌﾄﾓｰﾀｰ 正転(各個)
      AND     X0  ; 運転準備入り
      AND     M17  ; 運転ﾓｰﾄﾞ切替
      ANI     M104  ; 締め側ﾘﾌﾄﾓｰﾀｰ ｻｰﾏﾙﾄﾘｯﾌﾟ
      LD      M260  ; 締め部　ﾘﾌﾀｰ 　　上昇端
      OR      M261  ; 締め部　ﾘﾌﾀｰ 　　下降端
      ANB
      OUT     M686  ; 締め側　ﾘﾌﾄﾓｰﾀｰ 逆転(各個)
633   LD      M421  ; 連続運転
      LD      L200  ; 締め部　ﾘﾀｰﾝ⇒ﾘﾌﾀ ﾊﾟﾚｯﾄ通過中
      LD      Y2E6  ; 締め部　ﾘﾌﾀｰ 上昇SOL
      ANI     M260  ; 締め部　ﾘﾌﾀｰ 　　上昇端
      AND     T224  ; 締め部　ﾘﾌﾀｰ ﾊﾟﾚｯﾄ確認
      ORB
      ANB
      OR      M685  ; 締め側　ﾘﾌﾄﾓｰﾀｰ 正転(各個)
      LD      M300  ; 原点復帰PB
      OR      M301
      AND     L200  ; 締め部　ﾘﾀｰﾝ⇒ﾘﾌﾀ ﾊﾟﾚｯﾄ通過中
      ANI     L201  ; 締め部　ﾘﾀｰﾝ⇒ﾘﾌﾀ ﾊﾟﾚｯﾄ通過完了
      AND     M261  ; 締め部　ﾘﾌﾀｰ 　　下降端
      ORB
      OUT     Y8D  ; 締め側　ﾘﾌﾄﾓｰﾀｰ 正転
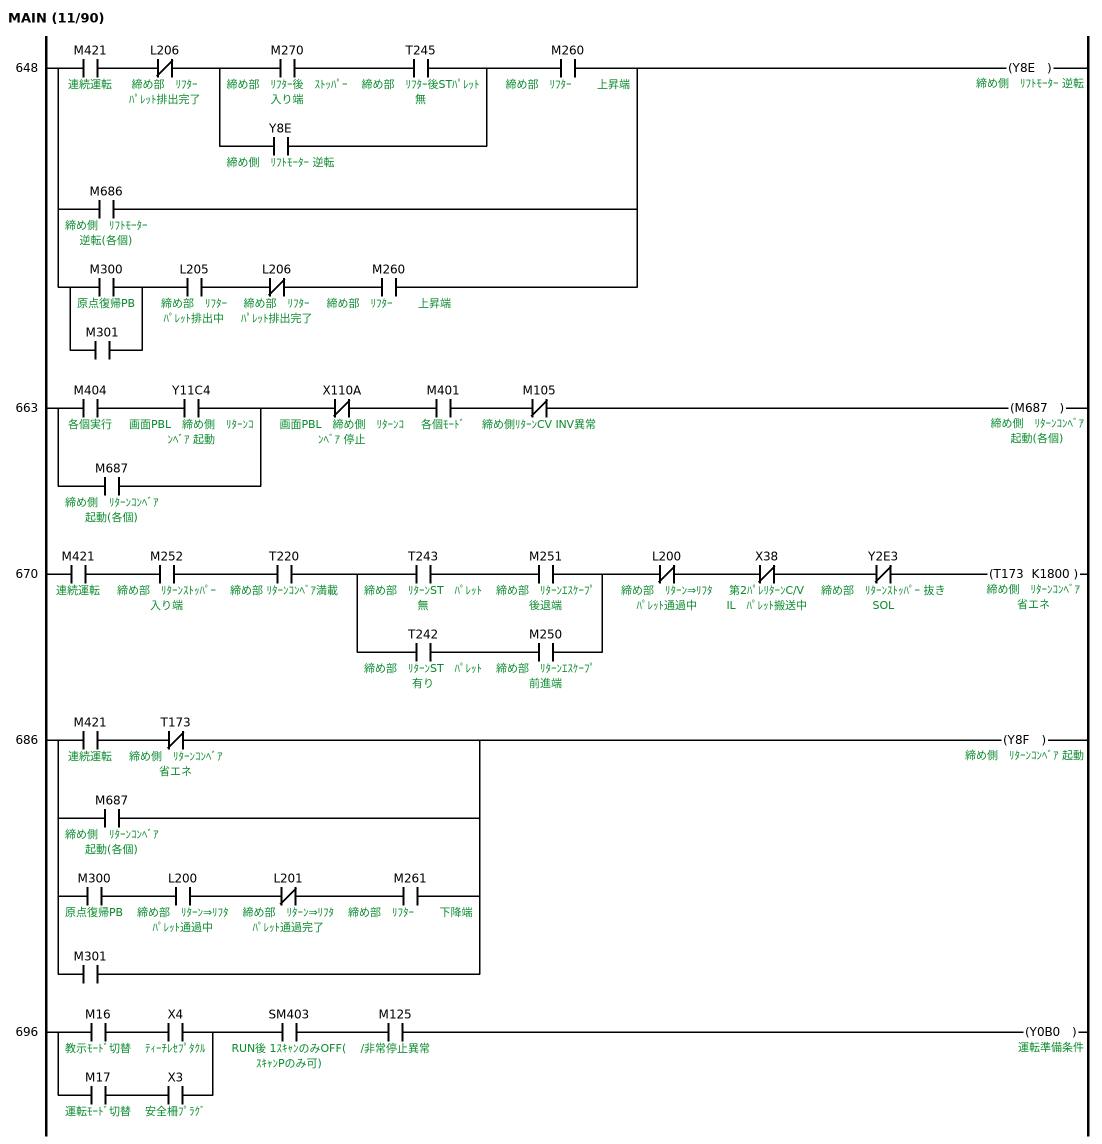
648   LD      M421  ; 連続運転
      ANI     L206  ; 締め部　ﾘﾌﾀｰ ﾊﾟﾚｯﾄ排出完了
      LD      M270  ; 締め部　ﾘﾌﾀｰ後　ｽﾄｯﾊﾟｰ　入り端
      AND     T245  ; 締め部　ﾘﾌﾀｰ後STﾊﾟﾚｯﾄ無
      OR      Y8E  ; 締め側　ﾘﾌﾄﾓｰﾀｰ 逆転
      ANB
      AND     M260  ; 締め部　ﾘﾌﾀｰ 　　上昇端
      OR      M686  ; 締め側　ﾘﾌﾄﾓｰﾀｰ 逆転(各個)
      LD      M300  ; 原点復帰PB
      OR      M301
      AND     L205  ; 締め部　ﾘﾌﾀｰ ﾊﾟﾚｯﾄ排出中
      ANI     L206  ; 締め部　ﾘﾌﾀｰ ﾊﾟﾚｯﾄ排出完了
      AND     M260  ; 締め部　ﾘﾌﾀｰ 　　上昇端
      ORB
      OUT     Y8E  ; 締め側　ﾘﾌﾄﾓｰﾀｰ 逆転
663   LD      M404  ; 各個実行
      AND     Y11C4  ; 画面PBL　締め側　ﾘﾀｰﾝｺﾝﾍﾞｱ 起動
      OR      M687  ; 締め側　ﾘﾀｰﾝｺﾝﾍﾞｱ 起動(各個)
      ANI     X110A  ; 画面PBL　締め側　ﾘﾀｰﾝｺﾝﾍﾞｱ 停止
      AND     M401  ; 各個ﾓｰﾄﾞ
      ANI     M105  ; 締め側ﾘﾀｰﾝCV INV異常
      OUT     M687  ; 締め側　ﾘﾀｰﾝｺﾝﾍﾞｱ 起動(各個)
670   LD      M421  ; 連続運転
      AND     M252  ; 締め部　ﾘﾀｰﾝｽﾄｯﾊﾟｰ 入り端
      AND     T220  ; 締め部 ﾘﾀｰﾝｺﾝﾍﾞｱ満載
      LD      T243  ; 締め部　ﾘﾀｰﾝST　ﾊﾟﾚｯﾄ無
      AND     M251  ; 締め部　ﾘﾀｰﾝｴｽｹｰﾌﾟ 後退端
      LD      T242  ; 締め部　ﾘﾀｰﾝST　ﾊﾟﾚｯﾄ有り
      AND     M250  ; 締め部　ﾘﾀｰﾝｴｽｹｰﾌﾟ 前進端
      ORB
      ANB
      ANI     L200  ; 締め部　ﾘﾀｰﾝ⇒ﾘﾌﾀ ﾊﾟﾚｯﾄ通過中
      ANI     X38  ; 第2ﾊﾟﾚﾘﾀｰﾝC/V IL　ﾊﾟﾚｯﾄ搬送中
      ANI     Y2E3  ; 締め部　ﾘﾀｰﾝｽﾄｯﾊﾟｰ 抜き SOL
      OUT     T173 K1800  ; 締め側　ﾘﾀｰﾝｺﾝﾍﾞｱ 省エネ
686   LD      M421  ; 連続運転
      ANI     T173  ; 締め側　ﾘﾀｰﾝｺﾝﾍﾞｱ 省エネ
      OR      M687  ; 締め側　ﾘﾀｰﾝｺﾝﾍﾞｱ 起動(各個)
      LD      M300  ; 原点復帰PB
      AND     L200  ; 締め部　ﾘﾀｰﾝ⇒ﾘﾌﾀ ﾊﾟﾚｯﾄ通過中
      ANI     L201  ; 締め部　ﾘﾀｰﾝ⇒ﾘﾌﾀ ﾊﾟﾚｯﾄ通過完了
      AND     M261  ; 締め部　ﾘﾌﾀｰ 　　下降端
      ORB
      OR      M301
      OUT     Y8F  ; 締め側　ﾘﾀｰﾝｺﾝﾍﾞｱ 起動
696   LD      M16  ; 教示ﾓｰﾄﾞ切替
      AND     X4  ; ﾃｨｰﾁﾚｾﾌﾟﾀｸﾙ
      LD      M17  ; 運転ﾓｰﾄﾞ切替
      AND     X3  ; 安全柵ﾌﾟﾗｸﾞ
      ORB
      AND     SM403  ; RUN後 1ｽｷｬﾝのみOFF(ｽｷｬﾝPのみ可)
      AND     M125  ; /非常停止異常
      OUT     Y0B0  ; 運転準備条件
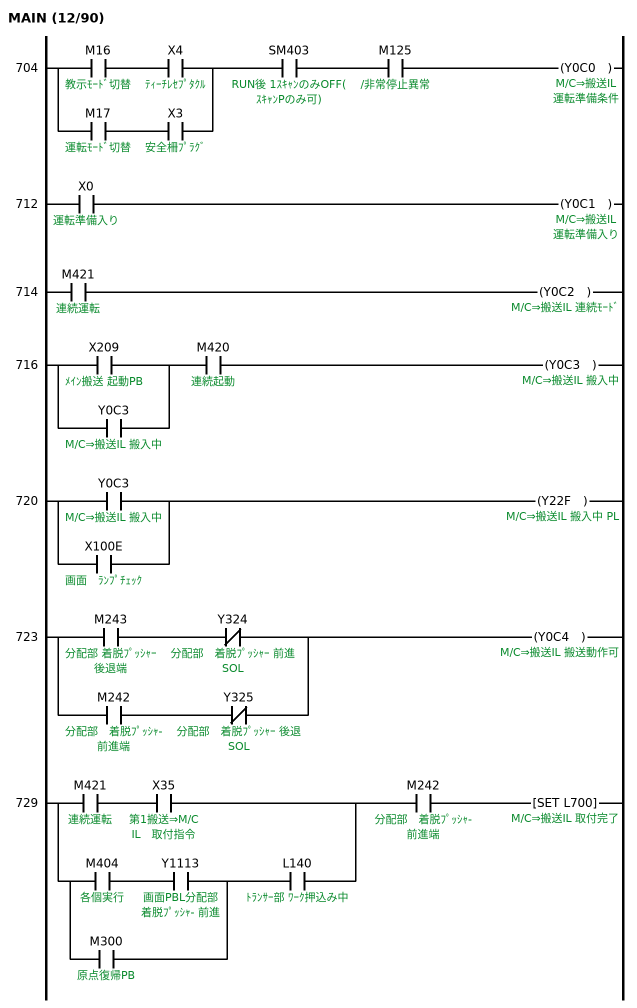
704   LD      M16  ; 教示ﾓｰﾄﾞ切替
      AND     X4  ; ﾃｨｰﾁﾚｾﾌﾟﾀｸﾙ
      LD      M17  ; 運転ﾓｰﾄﾞ切替
      AND     X3  ; 安全柵ﾌﾟﾗｸﾞ
      ORB
      AND     SM403  ; RUN後 1ｽｷｬﾝのみOFF(ｽｷｬﾝPのみ可)
      AND     M125  ; /非常停止異常
      OUT     Y0C0  ; M/C⇒搬送IL 運転準備条件
712   LD      X0  ; 運転準備入り
      OUT     Y0C1  ; M/C⇒搬送IL 運転準備入り
714   LD      M421  ; 連続運転
      OUT     Y0C2  ; M/C⇒搬送IL 連続ﾓｰﾄﾞ
716   LD      X209  ; ﾒｲﾝ搬送 起動PB
      OR      Y0C3  ; M/C⇒搬送IL 搬入中
      AND     M420  ; 連続起動
      OUT     Y0C3  ; M/C⇒搬送IL 搬入中
720   LD      Y0C3  ; M/C⇒搬送IL 搬入中
      OR      X100E  ; 画面　ﾗﾝﾌﾟﾁｪｯｸ
      OUT     Y22F  ; M/C⇒搬送IL 搬入中 PL
723   LD      M243  ; 分配部 着脱ﾌﾟｯｼｬｰ 後退端
      ANI     Y324  ; 分配部　着脱ﾌﾟｯｼｬｰ 前進 SOL
      LD      M242  ; 分配部　着脱ﾌﾟｯｼｬ- 前進端
      ANI     Y325  ; 分配部　着脱ﾌﾟｯｼｬｰ 後退 SOL
      ORB
      OUT     Y0C4  ; M/C⇒搬送IL 搬送動作可
729   LD      M421  ; 連続運転
      AND     X35  ; 第1搬送⇒M/C IL　取付指令
      LD      M404  ; 各個実行
      AND     Y1113  ; 画面PBL分配部 着脱ﾌﾟｯｼｬ- 前進
      OR      M300  ; 原点復帰PB
      AND     L140  ; ﾄﾗﾝｻｰ部 ﾜｰｸ押込み中
      ORB
      AND     M242  ; 分配部　着脱ﾌﾟｯｼｬ- 前進端
      SET     L700  ; M/C⇒搬送IL 取付完了
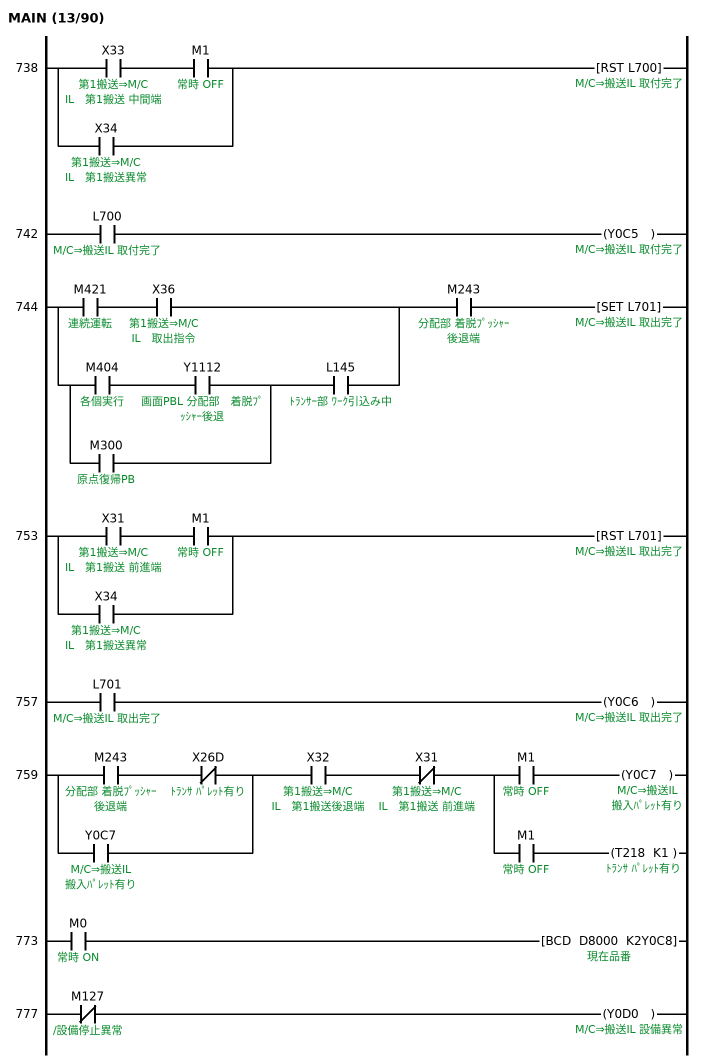
738   LD      X33  ; 第1搬送⇒M/C IL　第1搬送 中間端
      AND     M1  ; 常時 OFF
      OR      X34  ; 第1搬送⇒M/C IL　第1搬送異常
      RST     L700  ; M/C⇒搬送IL 取付完了
742   LD      L700  ; M/C⇒搬送IL 取付完了
      OUT     Y0C5  ; M/C⇒搬送IL 取付完了
744   LD      M421  ; 連続運転
      AND     X36  ; 第1搬送⇒M/C IL　取出指令
      LD      M404  ; 各個実行
      AND     Y1112  ; 画面PBL 分配部　着脱ﾌﾟｯｼｬｰ後退
      OR      M300  ; 原点復帰PB
      AND     L145  ; ﾄﾗﾝｻｰ部 ﾜｰｸ引込み中
      ORB
      AND     M243  ; 分配部 着脱ﾌﾟｯｼｬｰ 後退端
      SET     L701  ; M/C⇒搬送IL 取出完了
753   LD      X31  ; 第1搬送⇒M/C IL　第1搬送 前進端
      AND     M1  ; 常時 OFF
      OR      X34  ; 第1搬送⇒M/C IL　第1搬送異常
      RST     L701  ; M/C⇒搬送IL 取出完了
757   LD      L701  ; M/C⇒搬送IL 取出完了
      OUT     Y0C6  ; M/C⇒搬送IL 取出完了
759   LD      M243  ; 分配部 着脱ﾌﾟｯｼｬｰ 後退端
      ANI     X26D  ; ﾄﾗﾝｻ ﾊﾟﾚｯﾄ有り
      OR      Y0C7  ; M/C⇒搬送IL 搬入ﾊﾟﾚｯﾄ有り
      AND     X32  ; 第1搬送⇒M/C IL　第1搬送後退端
      ANI     X31  ; 第1搬送⇒M/C IL　第1搬送 前進端
      MPS
      AND     M1  ; 常時 OFF
      OUT     Y0C7  ; M/C⇒搬送IL 搬入ﾊﾟﾚｯﾄ有り
      MPP
      AND     M1  ; 常時 OFF
      OUT     T218 K1  ; ﾄﾗﾝｻ ﾊﾟﾚｯﾄ有り
773   LD      M0  ; 常時 ON
      BCD     D8000 K2Y0C8  ; 現在品番 / M/C⇒搬送IL ID情報 BCD01
777   LDI     M127  ; /設備停止異常
      OUT     Y0D0  ; M/C⇒搬送IL 設備異常
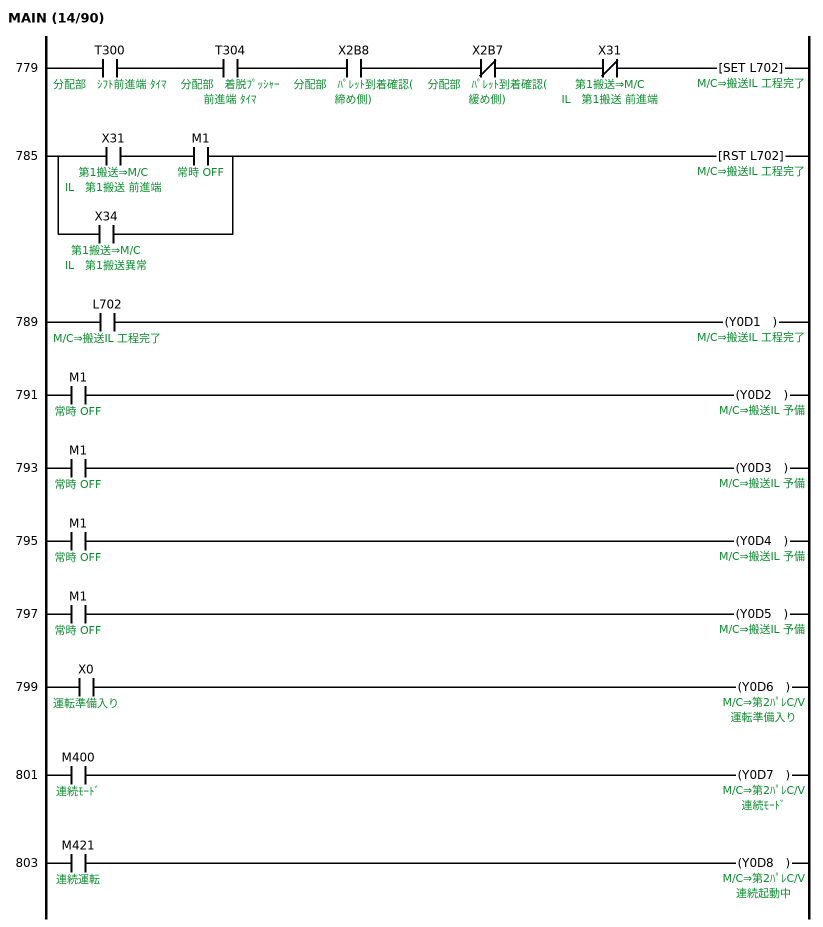
779   LD      T300  ; 分配部　ｼﾌﾄ前進端 ﾀｲﾏ
      AND     T304  ; 分配部　着脱ﾌﾟｯｼｬｰ 前進端 ﾀｲﾏ
      AND     X2B8  ; 分配部　ﾊﾟﾚｯﾄ到着確認(締め側)
      ANI     X2B7  ; 分配部　ﾊﾟﾚｯﾄ到着確認(緩め側)
      ANI     X31  ; 第1搬送⇒M/C IL　第1搬送 前進端
      SET     L702  ; M/C⇒搬送IL 工程完了
785   LD      X31  ; 第1搬送⇒M/C IL　第1搬送 前進端
      AND     M1  ; 常時 OFF
      OR      X34  ; 第1搬送⇒M/C IL　第1搬送異常
      RST     L702  ; M/C⇒搬送IL 工程完了
789   LD      L702  ; M/C⇒搬送IL 工程完了
      OUT     Y0D1  ; M/C⇒搬送IL 工程完了
791   LD      M1  ; 常時 OFF
      OUT     Y0D2  ; M/C⇒搬送IL 予備
793   LD      M1  ; 常時 OFF
      OUT     Y0D3  ; M/C⇒搬送IL 予備
795   LD      M1  ; 常時 OFF
      OUT     Y0D4  ; M/C⇒搬送IL 予備
797   LD      M1  ; 常時 OFF
      OUT     Y0D5  ; M/C⇒搬送IL 予備
799   LD      X0  ; 運転準備入り
      OUT     Y0D6  ; M/C⇒第2ﾊﾟﾚC/V 運転準備入り
801   LD      M400  ; 連続ﾓｰﾄﾞ
      OUT     Y0D7  ; M/C⇒第2ﾊﾟﾚC/V 連続ﾓｰﾄﾞ
803   LD      M421  ; 連続運転
      OUT     Y0D8  ; M/C⇒第2ﾊﾟﾚC/V 連続起動中
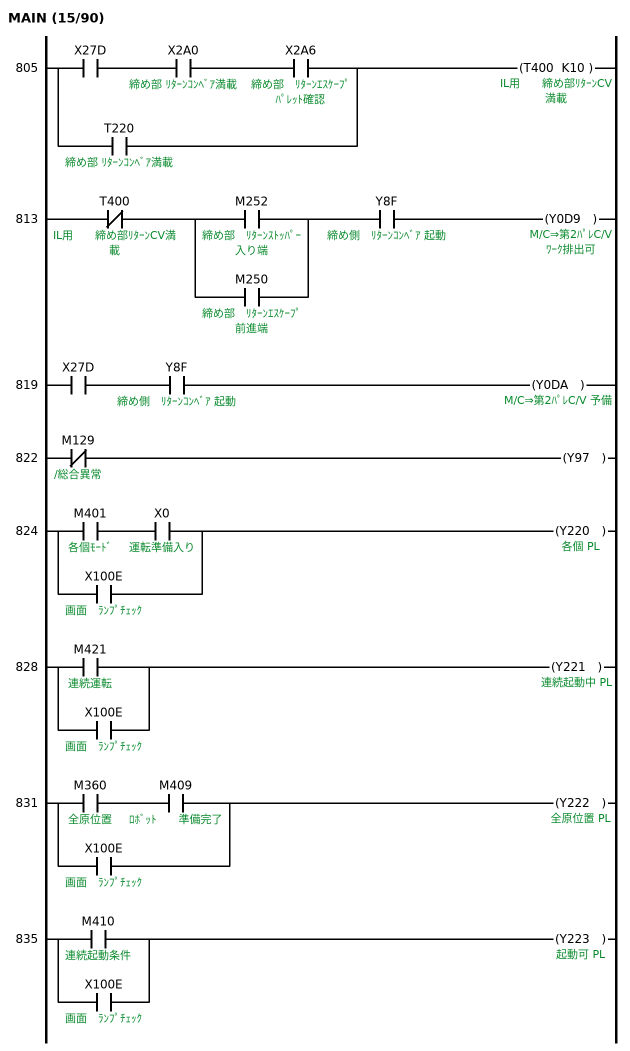
805   LD      X27D
      AND     X2A0  ; 締め部 ﾘﾀｰﾝｺﾝﾍﾞｱ満載
      AND     X2A6  ; 締め部　ﾘﾀｰﾝｴｽｹｰﾌﾟ ﾊﾟﾚｯﾄ確認
      OR      T220  ; 締め部 ﾘﾀｰﾝｺﾝﾍﾞｱ満載
      OUT     T400 K10  ; IL用　　締め部ﾘﾀｰﾝCV満載
813   LDI     T400  ; IL用　　締め部ﾘﾀｰﾝCV満載
      LD      M252  ; 締め部　ﾘﾀｰﾝｽﾄｯﾊﾟｰ 入り端
      OR      M250  ; 締め部　ﾘﾀｰﾝｴｽｹｰﾌﾟ 前進端
      ANB
      AND     Y8F  ; 締め側　ﾘﾀｰﾝｺﾝﾍﾞｱ 起動
      OUT     Y0D9  ; M/C⇒第2ﾊﾟﾚC/V ﾜｰｸ排出可
819   LD      X27D
      AND     Y8F  ; 締め側　ﾘﾀｰﾝｺﾝﾍﾞｱ 起動
      OUT     Y0DA  ; M/C⇒第2ﾊﾟﾚC/V 予備
822   LDI     M129  ; /総合異常
      OUT     Y97
824   LD      M401  ; 各個ﾓｰﾄﾞ
      AND     X0  ; 運転準備入り
      OR      X100E  ; 画面　ﾗﾝﾌﾟﾁｪｯｸ
      OUT     Y220  ; 各個 PL
828   LD      M421  ; 連続運転
      OR      X100E  ; 画面　ﾗﾝﾌﾟﾁｪｯｸ
      OUT     Y221  ; 連続起動中 PL
831   LD      M360  ; 全原位置
      AND     M409  ; ﾛﾎﾞｯﾄ　　準備完了
      OR      X100E  ; 画面　ﾗﾝﾌﾟﾁｪｯｸ
      OUT     Y222  ; 全原位置 PL
835   LD      M410  ; 連続起動条件
      OR      X100E  ; 画面　ﾗﾝﾌﾟﾁｪｯｸ
      OUT     Y223  ; 起動可 PL
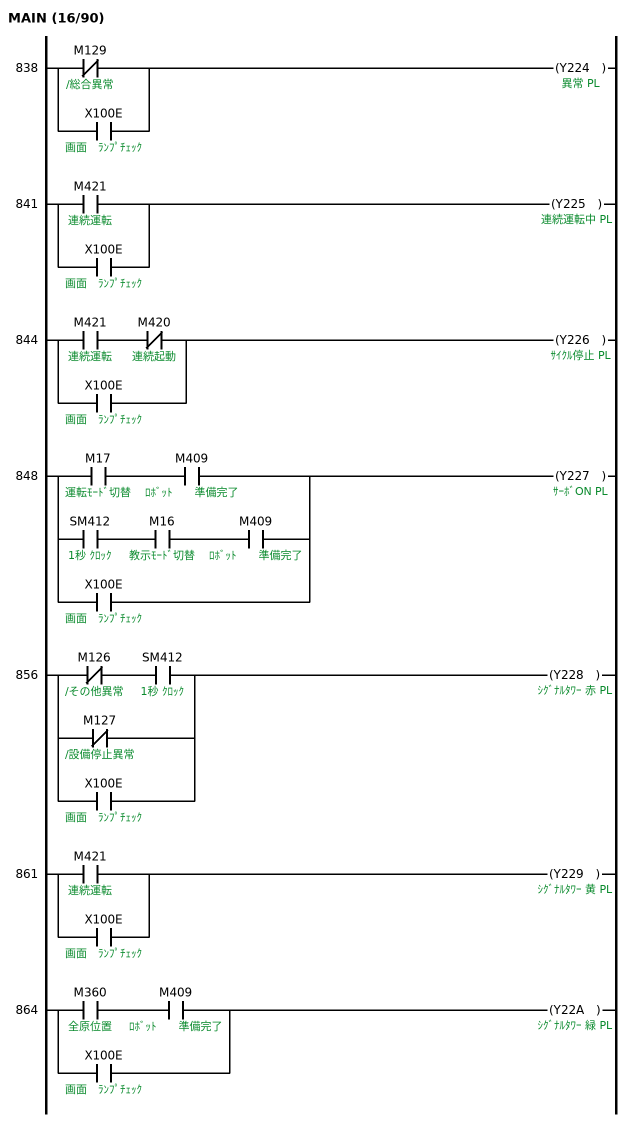
838   LDI     M129  ; /総合異常
      OR      X100E  ; 画面　ﾗﾝﾌﾟﾁｪｯｸ
      OUT     Y224  ; 異常 PL
841   LD      M421  ; 連続運転
      OR      X100E  ; 画面　ﾗﾝﾌﾟﾁｪｯｸ
      OUT     Y225  ; 連続運転中 PL
844   LD      M421  ; 連続運転
      ANI     M420  ; 連続起動
      OR      X100E  ; 画面　ﾗﾝﾌﾟﾁｪｯｸ
      OUT     Y226  ; ｻｲｸﾙ停止 PL
848   LD      M17  ; 運転ﾓｰﾄﾞ切替
      AND     M409  ; ﾛﾎﾞｯﾄ　　準備完了
      LD      SM412  ; 1秒 ｸﾛｯｸ
      AND     M16  ; 教示ﾓｰﾄﾞ切替
      AND     M409  ; ﾛﾎﾞｯﾄ　　準備完了
      ORB
      OR      X100E  ; 画面　ﾗﾝﾌﾟﾁｪｯｸ
      OUT     Y227  ; ｻｰﾎﾞON PL
856   LDI     M126  ; /その他異常
      AND     SM412  ; 1秒 ｸﾛｯｸ
      ORI     M127  ; /設備停止異常
      OR      X100E  ; 画面　ﾗﾝﾌﾟﾁｪｯｸ
      OUT     Y228  ; ｼｸﾞﾅﾙﾀﾜｰ 赤 PL
861   LD      M421  ; 連続運転
      OR      X100E  ; 画面　ﾗﾝﾌﾟﾁｪｯｸ
      OUT     Y229  ; ｼｸﾞﾅﾙﾀﾜｰ 黄 PL
864   LD      M360  ; 全原位置
      AND     M409  ; ﾛﾎﾞｯﾄ　　準備完了
      OR      X100E  ; 画面　ﾗﾝﾌﾟﾁｪｯｸ
      OUT     Y22A  ; ｼｸﾞﾅﾙﾀﾜｰ 緑 PL
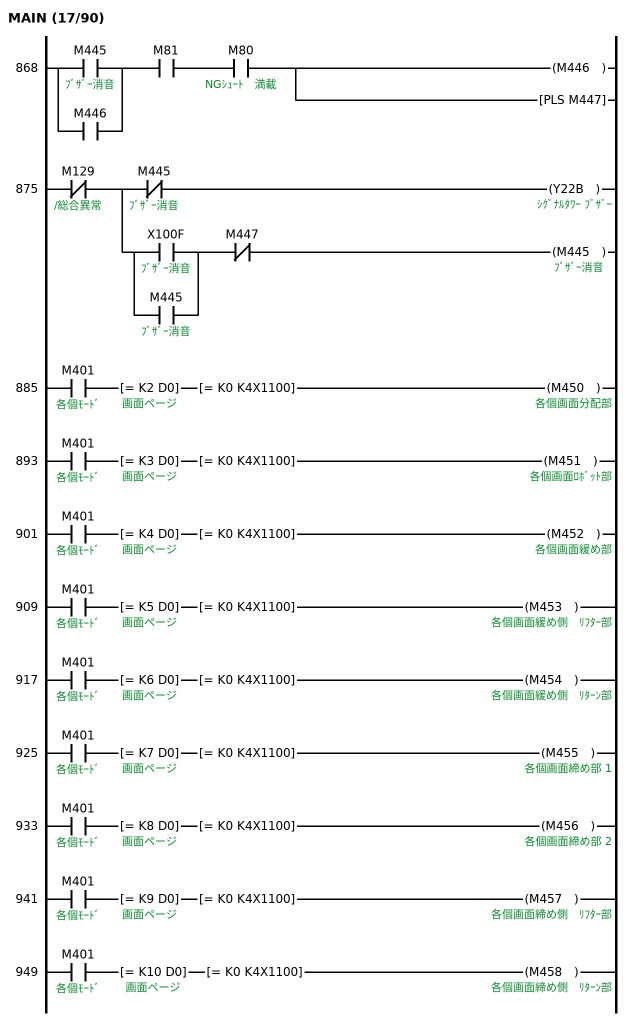
868   LD      M445  ; ﾌﾞｻﾞｰ消音
      OR      M446
      AND     M81
      AND     M80  ; NGｼｭｰﾄ　満載
      OUT     M446
      PLS     M447
875   LDI     M129  ; /総合異常
      MPS
      ANI     M445  ; ﾌﾞｻﾞｰ消音
      OUT     Y22B  ; ｼｸﾞﾅﾙﾀﾜｰ ﾌﾞｻﾞｰ
      MPP
      LD      X100F  ; ﾌﾞｻﾞｰ消音
      OR      M445  ; ﾌﾞｻﾞｰ消音
      ANB
      ANI     M447
      OUT     M445  ; ﾌﾞｻﾞｰ消音
885   LD      M401  ; 各個ﾓｰﾄﾞ
      AND=    K2 D0  ; 画面ページ
      AND=    K0 K4X1100  ; 画面PBL 緩め部　ﾒｲﾝ NR  停止
      OUT     M450  ; 各個画面分配部
893   LD      M401  ; 各個ﾓｰﾄﾞ
      AND=    K3 D0  ; 画面ページ
      AND=    K0 K4X1100  ; 画面PBL 緩め部　ﾒｲﾝ NR  停止
      OUT     M451  ; 各個画面ﾛﾎﾞｯﾄ部
901   LD      M401  ; 各個ﾓｰﾄﾞ
      AND=    K4 D0  ; 画面ページ
      AND=    K0 K4X1100  ; 画面PBL 緩め部　ﾒｲﾝ NR  停止
      OUT     M452  ; 各個画面緩め部
909   LD      M401  ; 各個ﾓｰﾄﾞ
      AND=    K5 D0  ; 画面ページ
      AND=    K0 K4X1100  ; 画面PBL 緩め部　ﾒｲﾝ NR  停止
      OUT     M453  ; 各個画面緩め側　ﾘﾌﾀｰ部
917   LD      M401  ; 各個ﾓｰﾄﾞ
      AND=    K6 D0  ; 画面ページ
      AND=    K0 K4X1100  ; 画面PBL 緩め部　ﾒｲﾝ NR  停止
      OUT     M454  ; 各個画面緩め側　ﾘﾀｰﾝ部
925   LD      M401  ; 各個ﾓｰﾄﾞ
      AND=    K7 D0  ; 画面ページ
      AND=    K0 K4X1100  ; 画面PBL 緩め部　ﾒｲﾝ NR  停止
      OUT     M455  ; 各個画面締め部 1
933   LD      M401  ; 各個ﾓｰﾄﾞ
      AND=    K8 D0  ; 画面ページ
      AND=    K0 K4X1100  ; 画面PBL 緩め部　ﾒｲﾝ NR  停止
      OUT     M456  ; 各個画面締め部 2
941   LD      M401  ; 各個ﾓｰﾄﾞ
      AND=    K9 D0  ; 画面ページ
      AND=    K0 K4X1100  ; 画面PBL 緩め部　ﾒｲﾝ NR  停止
      OUT     M457  ; 各個画面締め側　ﾘﾌﾀｰ部
949   LD      M401  ; 各個ﾓｰﾄﾞ
      AND=    K10 D0  ; 画面ページ
      AND=    K0 K4X1100  ; 画面PBL 緩め部　ﾒｲﾝ NR  停止
      OUT     M458  ; 各個画面締め側　ﾘﾀｰﾝ部
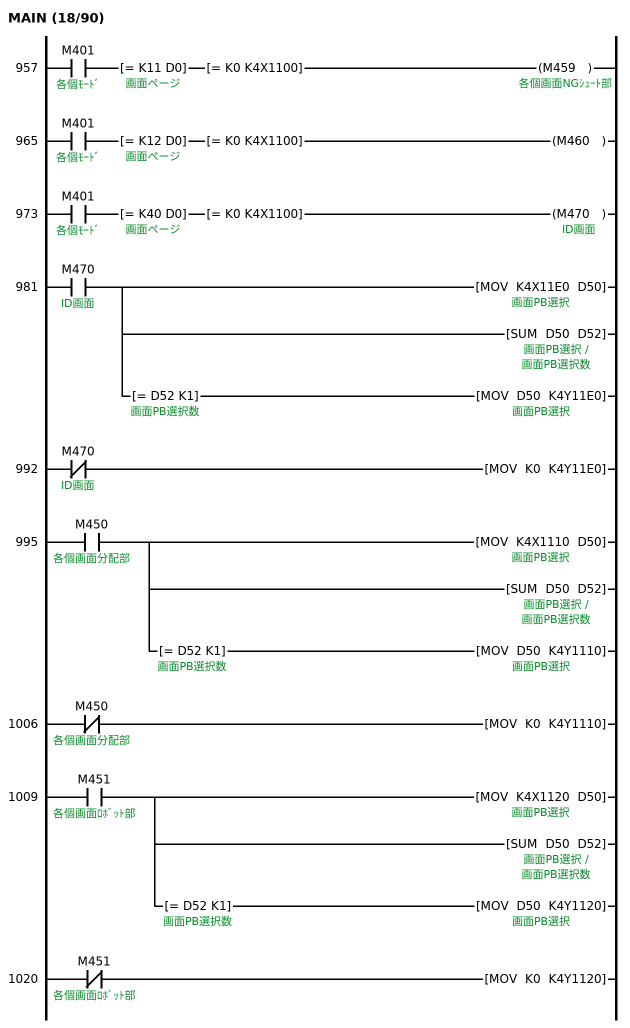
957   LD      M401  ; 各個ﾓｰﾄﾞ
      AND=    K11 D0  ; 画面ページ
      AND=    K0 K4X1100  ; 画面PBL 緩め部　ﾒｲﾝ NR  停止
      OUT     M459  ; 各個画面NGｼｭｰﾄ部
965   LD      M401  ; 各個ﾓｰﾄﾞ
      AND=    K12 D0  ; 画面ページ
      AND=    K0 K4X1100  ; 画面PBL 緩め部　ﾒｲﾝ NR  停止
      OUT     M460
973   LD      M401  ; 各個ﾓｰﾄﾞ
      AND=    K40 D0  ; 画面ページ
      AND=    K0 K4X1100  ; 画面PBL 緩め部　ﾒｲﾝ NR  停止
      OUT     M470  ; ID画面
981   LD      M470  ; ID画面
      MOV     K4X11E0 D50  ; 画面PBL / 画面PB選択
      SUM     D50 D52  ; 画面PB選択数
      AND=    D52 K1  ; 画面PB選択数
      MOV     D50 K4Y11E0  ; 画面PBL
992   LDI     M470  ; ID画面
      MOV     K0 K4Y11E0
995   LD      M450  ; 各個画面分配部
      MOV     K4X1110 D50  ; 画面PBL
      SUM     D50 D52
      AND=    D52 K1  ; 画面PB選択数
      MOV     D50 K4Y1110  ; 画面PBL分配部　ｼﾌﾄ 後退
1006  LDI     M450  ; 各個画面分配部
      MOV     K0 K4Y1110
1009  LD      M451  ; 各個画面ﾛﾎﾞｯﾄ部
      MOV     K4X1120 D50  ; 画面PBL
      SUM     D50 D52
      AND=    D52 K1  ; 画面PB選択数
      MOV     D50 K4Y1120  ; 画面PBL ﾛﾎﾞｯﾄﾁｬｯｸ開
1020  LDI     M451  ; 各個画面ﾛﾎﾞｯﾄ部
      MOV     K0 K4Y1120
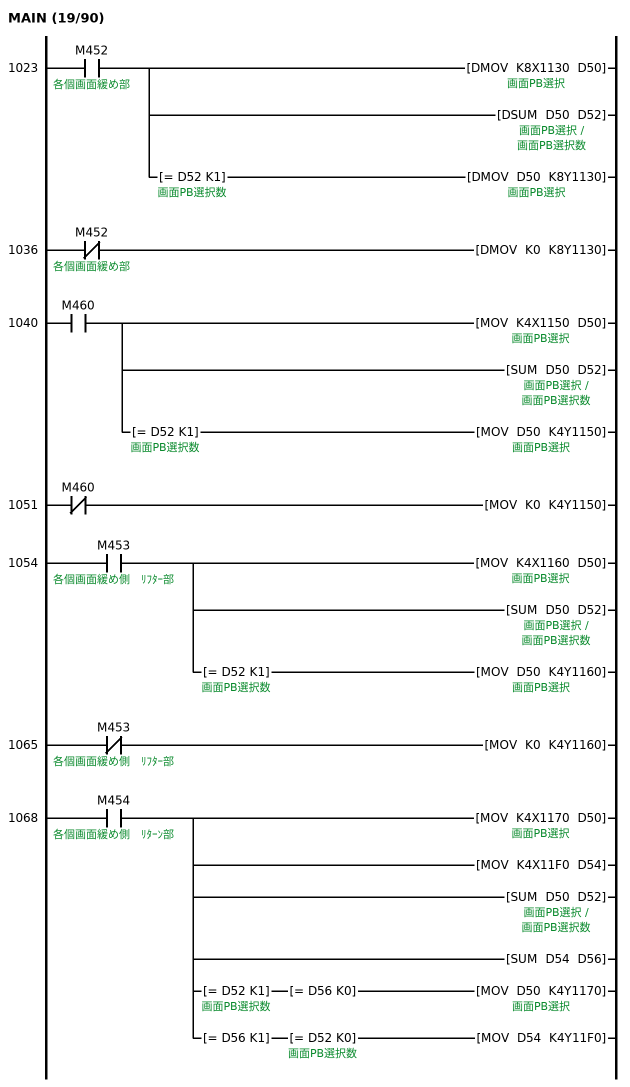
1023  LD      M452  ; 各個画面緩め部
      DMOV    K8X1130 D50  ; 画面PBL
      DSUM    D50 D52
      AND=    D52 K1  ; 画面PB選択数
      DMOV    D50 K8Y1130  ; 画面PBL緩め部 押込み 後退
1036  LDI     M452  ; 各個画面緩め部
      DMOV    K0 K8Y1130
1040  LD      M460
      MOV     K4X1150 D50  ; 画面PBL
      SUM     D50 D52
      AND=    D52 K1  ; 画面PB選択数
      MOV     D50 K4Y1150  ; 画面PBL　緩め部　ﾒｲﾝ NR  下降
1051  LDI     M460
      MOV     K0 K4Y1150
1054  LD      M453  ; 各個画面緩め側　ﾘﾌﾀｰ部
      MOV     K4X1160 D50  ; 画面PBL
      SUM     D50 D52
      AND=    D52 K1  ; 画面PB選択数
      MOV     D50 K4Y1160  ; 画面PBL緩め部　ﾘﾌﾀｰ 下降
1065  LDI     M453  ; 各個画面緩め側　ﾘﾌﾀｰ部
      MOV     K0 K4Y1160
1068  LD      M454  ; 各個画面緩め側　ﾘﾀｰﾝ部
      MOV     K4X1170 D50  ; 画面PBL
      MOV     K4X11F0 D54  ; 画面PBL
      SUM     D50 D52
      SUM     D54 D56
      MPS
      AND=    D52 K1  ; 画面PB選択数
      AND=    D56 K0
      MOV     D50 K4Y1170  ; 画面PBL緩め部　ﾘﾀｰﾝｴｽｹｰﾌﾟ 後退
      MPP
      AND=    D56 K1
      AND=    D52 K0  ; 画面PB選択数
      MOV     D54 K4Y11F0
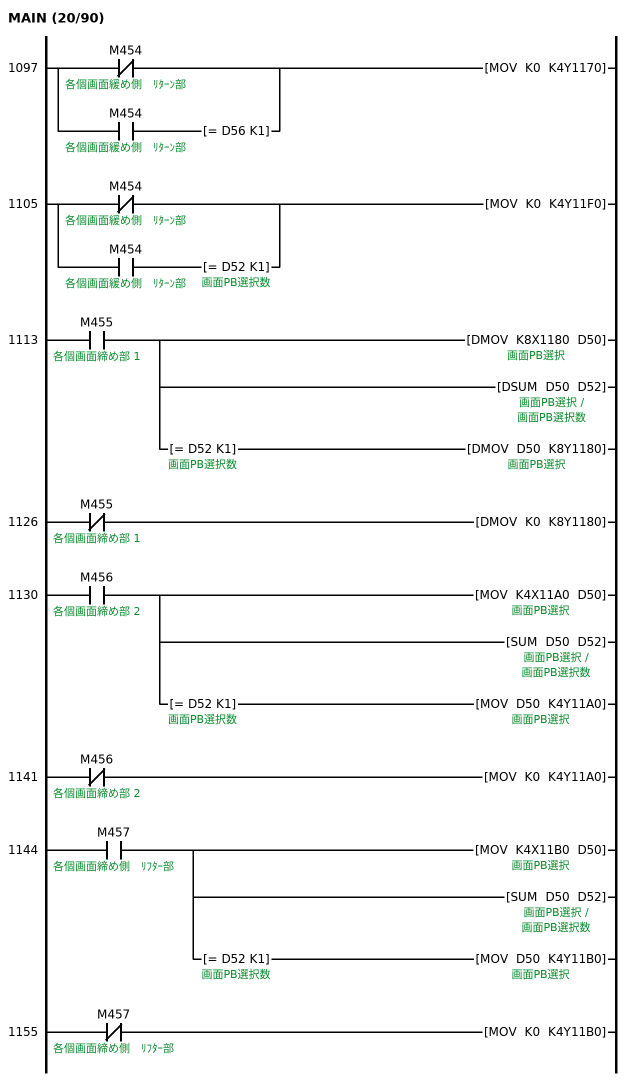
1097  LDI     M454  ; 各個画面緩め側　ﾘﾀｰﾝ部
      LD      M454  ; 各個画面緩め側　ﾘﾀｰﾝ部
      AND=    D56 K1
      ORB
      MOV     K0 K4Y1170
1105  LDI     M454  ; 各個画面緩め側　ﾘﾀｰﾝ部
      LD      M454  ; 各個画面緩め側　ﾘﾀｰﾝ部
      AND=    D52 K1  ; 画面PB選択数
      ORB
      MOV     K0 K4Y11F0
1113  LD      M455  ; 各個画面締め部 1
      DMOV    K8X1180 D50  ; 画面PBL
      DSUM    D50 D52
      AND=    D52 K1  ; 画面PB選択数
      DMOV    D50 K8Y1180  ; 画面PBL締め部　ﾘﾌﾀｰ後ｽﾄｯﾊﾟｰ抜き
1126  LDI     M455  ; 各個画面締め部 1
      DMOV    K0 K8Y1180
1130  LD      M456  ; 各個画面締め部 2
      MOV     K4X11A0 D50  ; 画面PBL
      SUM     D50 D52
      AND=    D52 K1  ; 画面PB選択数
      MOV     D50 K4Y11A0  ; 画面PBL　締め部　ﾅｯﾄﾗﾝﾅｰ 下降
1141  LDI     M456  ; 各個画面締め部 2
      MOV     K0 K4Y11A0
1144  LD      M457  ; 各個画面締め側　ﾘﾌﾀｰ部
      MOV     K4X11B0 D50  ; 画面PBL
      SUM     D50 D52
      AND=    D52 K1  ; 画面PB選択数
      MOV     D50 K4Y11B0  ; 画面PBL締め部　ﾘﾌﾀｰ 下降
1155  LDI     M457  ; 各個画面締め側　ﾘﾌﾀｰ部
      MOV     K0 K4Y11B0
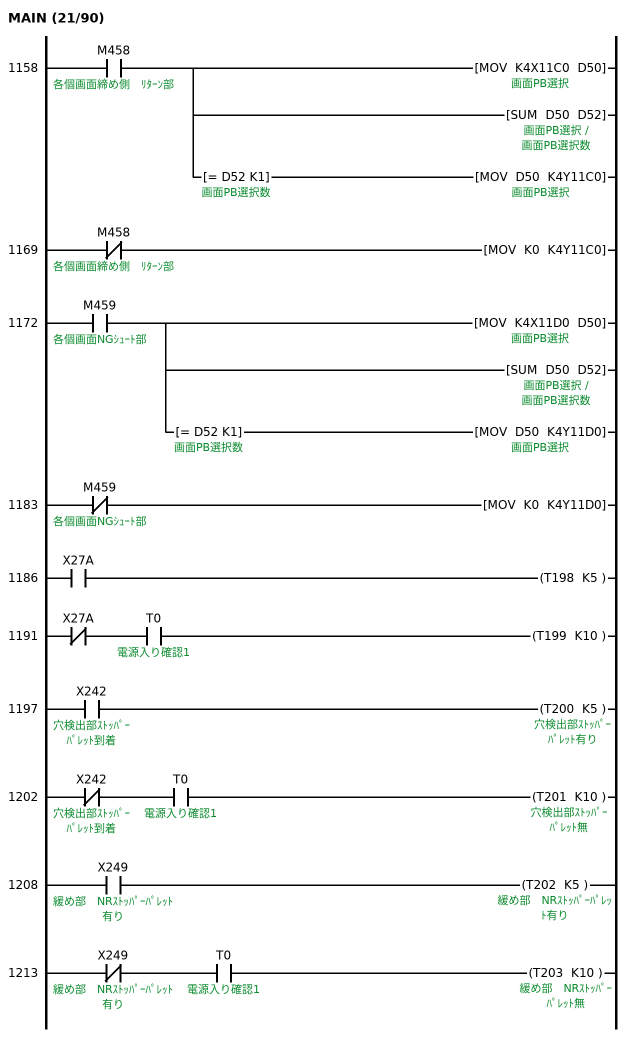
1158  LD      M458  ; 各個画面締め側　ﾘﾀｰﾝ部
      MOV     K4X11C0 D50  ; 画面PBL
      SUM     D50 D52
      AND=    D52 K1  ; 画面PB選択数
      MOV     D50 K4Y11C0  ; 画面PBL締め部　ﾘﾀｰﾝｴｽｹｰﾌﾟ 後退
1169  LDI     M458  ; 各個画面締め側　ﾘﾀｰﾝ部
      MOV     K0 K4Y11C0
1172  LD      M459  ; 各個画面NGｼｭｰﾄ部
      MOV     K4X11D0 D50  ; 画面PBL
      SUM     D50 D52
      AND=    D52 K1  ; 画面PB選択数
      MOV     D50 K4Y11D0  ; 画面PBL NGﾘﾌﾀｰ　下降
1183  LDI     M459  ; 各個画面NGｼｭｰﾄ部
      MOV     K0 K4Y11D0
1186  LD      X27A
      OUT     T198 K5
1191  LDI     X27A
      AND     T0  ; 電源入り確認1
      OUT     T199 K10
1197  LD      X242  ; 穴検出部ｽﾄｯﾊﾟｰ 　ﾊﾟﾚｯﾄ到着
      OUT     T200 K5  ; 穴検出部ｽﾄｯﾊﾟｰ 　ﾊﾟﾚｯﾄ有り
1202  LDI     X242  ; 穴検出部ｽﾄｯﾊﾟｰ 　ﾊﾟﾚｯﾄ到着
      AND     T0  ; 電源入り確認1
      OUT     T201 K10  ; 穴検出部ｽﾄｯﾊﾟｰ 　ﾊﾟﾚｯﾄ無
1208  LD      X249  ; 緩め部　NRｽﾄｯﾊﾟｰﾊﾟﾚｯﾄ有り
      OUT     T202 K5  ; 緩め部　NRｽﾄｯﾊﾟｰﾊﾟﾚｯﾄ有り
1213  LDI     X249  ; 緩め部　NRｽﾄｯﾊﾟｰﾊﾟﾚｯﾄ有り
      AND     T0  ; 電源入り確認1
      OUT     T203 K10  ; 緩め部　NRｽﾄｯﾊﾟｰ ﾊﾟﾚｯﾄ無
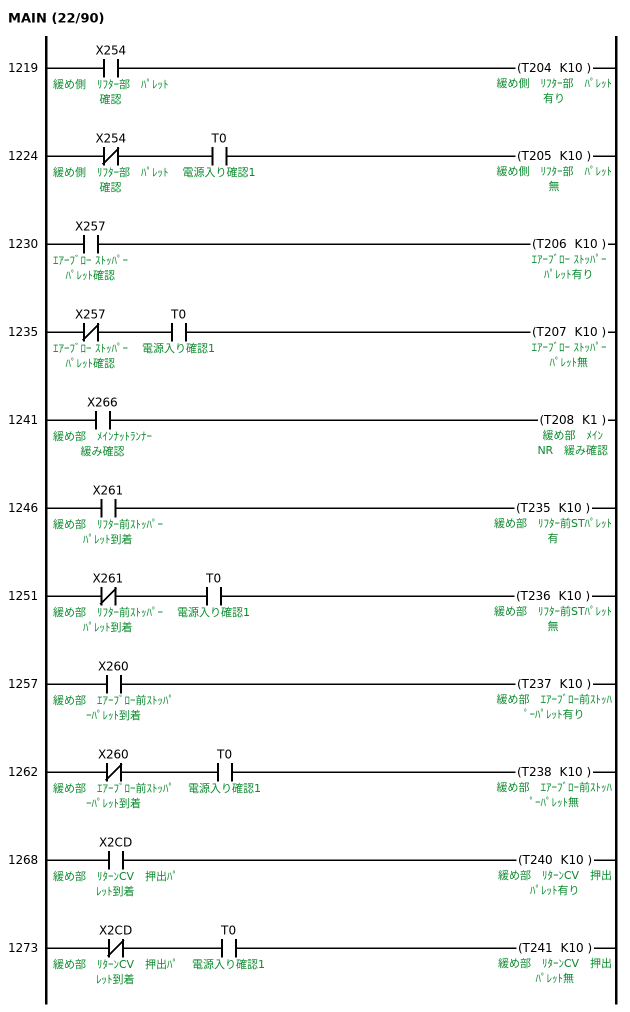
1219  LD      X254  ; 緩め側　ﾘﾌﾀｰ部　ﾊﾟﾚｯﾄ確認
      OUT     T204 K10  ; 緩め側　ﾘﾌﾀｰ部　ﾊﾟﾚｯﾄ有り
1224  LDI     X254  ; 緩め側　ﾘﾌﾀｰ部　ﾊﾟﾚｯﾄ確認
      AND     T0  ; 電源入り確認1
      OUT     T205 K10  ; 緩め側　ﾘﾌﾀｰ部　ﾊﾟﾚｯﾄ無
1230  LD      X257  ; ｴｱｰﾌﾞﾛｰ ｽﾄｯﾊﾟｰ  ﾊﾟﾚｯﾄ確認
      OUT     T206 K10  ; ｴｱｰﾌﾞﾛｰ ｽﾄｯﾊﾟｰ  ﾊﾟﾚｯﾄ有り
1235  LDI     X257  ; ｴｱｰﾌﾞﾛｰ ｽﾄｯﾊﾟｰ  ﾊﾟﾚｯﾄ確認
      AND     T0  ; 電源入り確認1
      OUT     T207 K10  ; ｴｱｰﾌﾞﾛｰ ｽﾄｯﾊﾟｰ  ﾊﾟﾚｯﾄ無
1241  LD      X266  ; 緩め部　ﾒｲﾝﾅｯﾄﾗﾝﾅｰ 緩み確認
      OUT     T208 K1  ; 緩め部　ﾒｲﾝ NR　緩み確認
1246  LD      X261  ; 緩め部　ﾘﾌﾀｰ前ｽﾄｯﾊﾟｰ　ﾊﾟﾚｯﾄ到着
      OUT     T235 K10  ; 緩め部　ﾘﾌﾀｰ前STﾊﾟﾚｯﾄ有
1251  LDI     X261  ; 緩め部　ﾘﾌﾀｰ前ｽﾄｯﾊﾟｰ　ﾊﾟﾚｯﾄ到着
      AND     T0  ; 電源入り確認1
      OUT     T236 K10  ; 緩め部　ﾘﾌﾀｰ前STﾊﾟﾚｯﾄ無
1257  LD      X260  ; 緩め部　ｴｱｰﾌﾞﾛｰ前ｽﾄｯﾊﾟｰﾊﾟﾚｯﾄ到着
      OUT     T237 K10  ; 緩め部　ｴｱｰﾌﾞﾛｰ前ｽﾄｯﾊﾟｰﾊﾟﾚｯﾄ有り
1262  LDI     X260  ; 緩め部　ｴｱｰﾌﾞﾛｰ前ｽﾄｯﾊﾟｰﾊﾟﾚｯﾄ到着
      AND     T0  ; 電源入り確認1
      OUT     T238 K10  ; 緩め部　ｴｱｰﾌﾞﾛｰ前ｽﾄｯﾊﾟｰﾊﾟﾚｯﾄ無
1268  LD      X2CD  ; 緩め部　ﾘﾀｰﾝCV　押出ﾊﾟﾚｯﾄ到着
      OUT     T240 K10  ; 緩め部　ﾘﾀｰﾝCV　押出ﾊﾟﾚｯﾄ有り
1273  LDI     X2CD  ; 緩め部　ﾘﾀｰﾝCV　押出ﾊﾟﾚｯﾄ到着
      AND     T0  ; 電源入り確認1
      OUT     T241 K10  ; 緩め部　ﾘﾀｰﾝCV　押出ﾊﾟﾚｯﾄ無
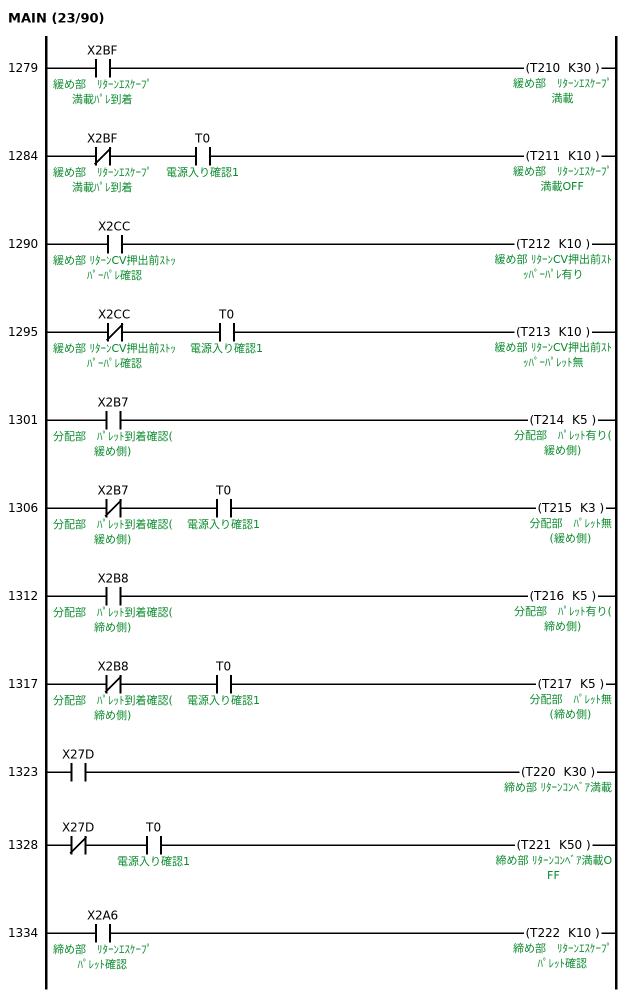
1279  LD      X2BF  ; 緩め部　ﾘﾀｰﾝｴｽｹｰﾌﾟ 満載ﾊﾟﾚ到着
      OUT     T210 K30  ; 緩め部　ﾘﾀｰﾝｴｽｹｰﾌﾟ 満載
1284  LDI     X2BF  ; 緩め部　ﾘﾀｰﾝｴｽｹｰﾌﾟ 満載ﾊﾟﾚ到着
      AND     T0  ; 電源入り確認1
      OUT     T211 K10  ; 緩め部　ﾘﾀｰﾝｴｽｹｰﾌﾟ 満載OFF
1290  LD      X2CC  ; 緩め部 ﾘﾀｰﾝCV押出前ｽﾄｯﾊﾟｰﾊﾟﾚ確認
      OUT     T212 K10  ; 緩め部 ﾘﾀｰﾝCV押出前ｽﾄｯﾊﾟｰﾊﾟﾚ有り
1295  LDI     X2CC  ; 緩め部 ﾘﾀｰﾝCV押出前ｽﾄｯﾊﾟｰﾊﾟﾚ確認
      AND     T0  ; 電源入り確認1
      OUT     T213 K10  ; 緩め部 ﾘﾀｰﾝCV押出前ｽﾄｯﾊﾟｰﾊﾟﾚｯﾄ無
1301  LD      X2B7  ; 分配部　ﾊﾟﾚｯﾄ到着確認(緩め側)
      OUT     T214 K5  ; 分配部　ﾊﾟﾚｯﾄ有り(緩め側)
1306  LDI     X2B7  ; 分配部　ﾊﾟﾚｯﾄ到着確認(緩め側)
      AND     T0  ; 電源入り確認1
      OUT     T215 K3  ; 分配部　ﾊﾟﾚｯﾄ無 (緩め側)
1312  LD      X2B8  ; 分配部　ﾊﾟﾚｯﾄ到着確認(締め側)
      OUT     T216 K5  ; 分配部　ﾊﾟﾚｯﾄ有り(締め側)
1317  LDI     X2B8  ; 分配部　ﾊﾟﾚｯﾄ到着確認(締め側)
      AND     T0  ; 電源入り確認1
      OUT     T217 K5  ; 分配部　ﾊﾟﾚｯﾄ無 (締め側)
1323  LD      X27D
      OUT     T220 K30  ; 締め部 ﾘﾀｰﾝｺﾝﾍﾞｱ満載
1328  LDI     X27D
      AND     T0  ; 電源入り確認1
      OUT     T221 K50  ; 締め部 ﾘﾀｰﾝｺﾝﾍﾞｱ満載OFF
1334  LD      X2A6  ; 締め部　ﾘﾀｰﾝｴｽｹｰﾌﾟ ﾊﾟﾚｯﾄ確認
      OUT     T222 K10  ; 締め部　ﾘﾀｰﾝｴｽｹｰﾌﾟ ﾊﾟﾚｯﾄ確認
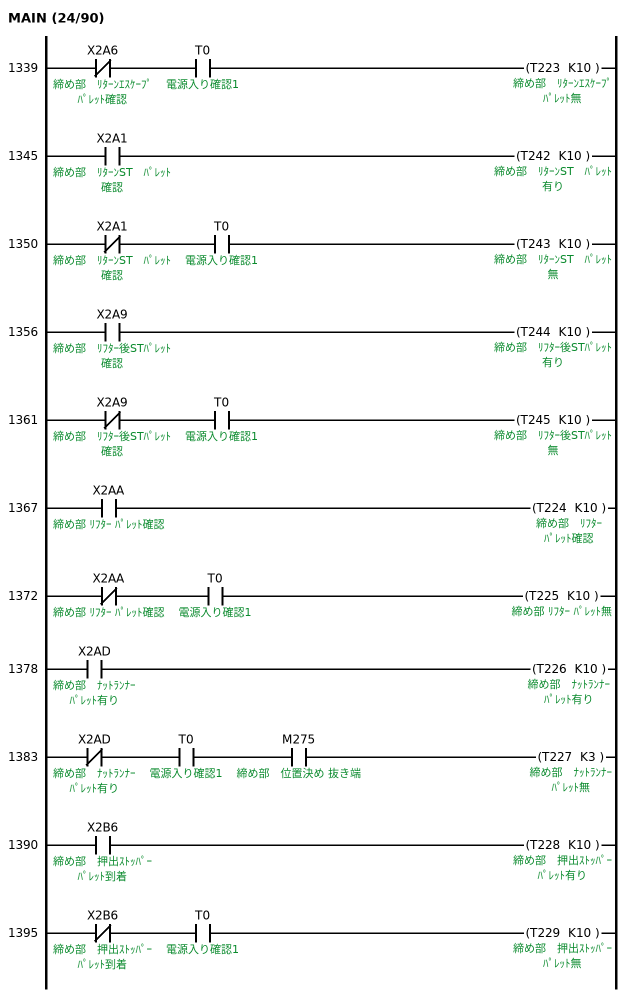
1339  LDI     X2A6  ; 締め部　ﾘﾀｰﾝｴｽｹｰﾌﾟ ﾊﾟﾚｯﾄ確認
      AND     T0  ; 電源入り確認1
      OUT     T223 K10  ; 締め部　ﾘﾀｰﾝｴｽｹｰﾌﾟ ﾊﾟﾚｯﾄ無
1345  LD      X2A1  ; 締め部　ﾘﾀｰﾝST　ﾊﾟﾚｯﾄ確認
      OUT     T242 K10  ; 締め部　ﾘﾀｰﾝST　ﾊﾟﾚｯﾄ有り
1350  LDI     X2A1  ; 締め部　ﾘﾀｰﾝST　ﾊﾟﾚｯﾄ確認
      AND     T0  ; 電源入り確認1
      OUT     T243 K10  ; 締め部　ﾘﾀｰﾝST　ﾊﾟﾚｯﾄ無
1356  LD      X2A9  ; 締め部　ﾘﾌﾀｰ後STﾊﾟﾚｯﾄ確認
      OUT     T244 K10  ; 締め部　ﾘﾌﾀｰ後STﾊﾟﾚｯﾄ有り
1361  LDI     X2A9  ; 締め部　ﾘﾌﾀｰ後STﾊﾟﾚｯﾄ確認
      AND     T0  ; 電源入り確認1
      OUT     T245 K10  ; 締め部　ﾘﾌﾀｰ後STﾊﾟﾚｯﾄ無
1367  LD      X2AA  ; 締め部 ﾘﾌﾀｰ ﾊﾟﾚｯﾄ確認
      OUT     T224 K10  ; 締め部　ﾘﾌﾀｰ ﾊﾟﾚｯﾄ確認
1372  LDI     X2AA  ; 締め部 ﾘﾌﾀｰ ﾊﾟﾚｯﾄ確認
      AND     T0  ; 電源入り確認1
      OUT     T225 K10  ; 締め部 ﾘﾌﾀｰ ﾊﾟﾚｯﾄ無
1378  LD      X2AD  ; 締め部　ﾅｯﾄﾗﾝﾅｰ ﾊﾟﾚｯﾄ有り
      OUT     T226 K10  ; 締め部　ﾅｯﾄﾗﾝﾅｰ ﾊﾟﾚｯﾄ有り
1383  LDI     X2AD  ; 締め部　ﾅｯﾄﾗﾝﾅｰ ﾊﾟﾚｯﾄ有り
      AND     T0  ; 電源入り確認1
      AND     M275  ; 締め部　位置決め 抜き端
      OUT     T227 K3  ; 締め部　ﾅｯﾄﾗﾝﾅｰ ﾊﾟﾚｯﾄ無
1390  LD      X2B6  ; 締め部　押出ｽﾄｯﾊﾟｰ ﾊﾟﾚｯﾄ到着
      OUT     T228 K10  ; 締め部　押出ｽﾄｯﾊﾟｰ ﾊﾟﾚｯﾄ有り
1395  LDI     X2B6  ; 締め部　押出ｽﾄｯﾊﾟｰ ﾊﾟﾚｯﾄ到着
      AND     T0  ; 電源入り確認1
      OUT     T229 K10  ; 締め部　押出ｽﾄｯﾊﾟｰ ﾊﾟﾚｯﾄ無
